    movel([0.126018, -1.331569, -2.603647, -0.777173, 1.570796, 1.696815],accel_mss,speed_ms,0,blend_radius_m)
    movel([0.125748, -1.331456, -2.603719, -0.777214, 1.570796, 1.696544],accel_mss,speed_ms,0,blend_radius_m)
    movel([0.125813, -1.331140, -2.603920, -0.777329, 1.570796, 1.696609],accel_mss,speed_ms,0,blend_radius_m)
    movel([0.126327, -1.330807, -2.604132, -0.777450, 1.570796, 1.697124],accel_mss,speed_ms,0,blend_radius_m)
    movel([0.126943, -1.330606, -2.604260, -0.777523, 1.570796, 1.697739],accel_mss,speed_ms,0,blend_radius_m)
    movel([0.128465, -1.330173, -2.604536, -0.777680, 1.570796, 1.699261],accel_mss,speed_ms,0,blend_radius_m)
    speed_ms = 0.003
    movel([0.128465, -1.333596, -2.606105, -0.772688, 1.570796, 1.699261],accel_mss,speed_ms,0,blend_radius_m)
    speed_ms = 0.007
    movel([0.130070, -1.333157, -2.606385, -0.772846, 1.570796, 1.700866],accel_mss,speed_ms,0,blend_radius_m)
    movel([0.130779, -1.333015, -2.606476, -0.772898, 1.570796, 1.701575],accel_mss,speed_ms,0,blend_radius_m)
    movel([0.131107, -1.333043, -2.606458, -0.772888, 1.570796, 1.701903],accel_mss,speed_ms,0,blend_radius_m)
    movel([0.131205, -1.333224, -2.606343, -0.772822, 1.570796, 1.702001],accel_mss,speed_ms,0,blend_radius_m)
    movel([0.131006, -1.333538, -2.606142, -0.772709, 1.570796, 1.701802],accel_mss,speed_ms,0,blend_radius_m)
    movel([0.130299, -1.333839, -2.605950, -0.772600, 1.570796, 1.701096],accel_mss,speed_ms,0,blend_radius_m)
    movel([0.129539, -1.334076, -2.605798, -0.772515, 1.570796, 1.700335],accel_mss,speed_ms,0,blend_radius_m)
    movel([0.128417, -1.334397, -2.605593, -0.772399, 1.570796, 1.699213],accel_mss,speed_ms,0,blend_radius_m)
    movel([0.127106, -1.334758, -2.605362, -0.772269, 1.570796, 1.697903],accel_mss,speed_ms,0,blend_radius_m)
    movel([0.126423, -1.334924, -2.605256, -0.772210, 1.570796, 1.697219],accel_mss,speed_ms,0,blend_radius_m)
    movel([0.126018, -1.334988, -2.605214, -0.772187, 1.570796, 1.696815],accel_mss,speed_ms,0,blend_radius_m)
    movel([0.125748, -1.334876, -2.605286, -0.772227, 1.570796, 1.696544],accel_mss,speed_ms,0,blend_radius_m)
    movel([0.125813, -1.334561, -2.605488, -0.772340, 1.570796, 1.696609],accel_mss,speed_ms,0,blend_radius_m)
    movel([0.126327, -1.334229, -2.605700, -0.772460, 1.570796, 1.697124],accel_mss,speed_ms,0,blend_radius_m)
    movel([0.126943, -1.334028, -2.605829, -0.772532, 1.570796, 1.697739],accel_mss,speed_ms,0,blend_radius_m)
    movel([0.128465, -1.333596, -2.606105, -0.772688, 1.570796, 1.699261],accel_mss,speed_ms,0,blend_radius_m)
    speed_ms = 0.003
    movel([0.128465, -1.320057, -2.599778, -0.792554, 1.570796, 1.699261],accel_mss,speed_ms,0,blend_radius_m)
    speed_ms = 1.000
    movel([0.128465, -1.294201, -2.586731, -0.831457, 1.570796, 1.699261],accel_mss,speed_ms,0,blend_radius_m)
    movel([0.128376, -1.295380, -2.586019, -0.830991, 1.570796, 1.699172],accel_mss,speed_ms,0,blend_radius_m)
    movel([0.128376, -1.321218, -2.599050, -0.792121, 1.570796, 1.699172],accel_mss,speed_ms,0,blend_radius_m)
    speed_ms = 0.003
    movel([0.128376, -1.331325, -2.603802, -0.777262, 1.570796, 1.699172],accel_mss,speed_ms,0,blend_radius_m)
    speed_ms = 0.007
    movel([0.129253, -1.331084, -2.603956, -0.777349, 1.570796, 1.700049],accel_mss,speed_ms,0,blend_radius_m)
    movel([0.130004, -1.330891, -2.604079, -0.777419, 1.570796, 1.700800],accel_mss,speed_ms,0,blend_radius_m)
    movel([0.130651, -1.330733, -2.604179, -0.777477, 1.570796, 1.701447],accel_mss,speed_ms,0,blend_radius_m)
    movel([0.130767, -1.330971, -2.604028, -0.777390, 1.570796, 1.701564],accel_mss,speed_ms,0,blend_radius_m)
    movel([0.130518, -1.331302, -2.603817, -0.777270, 1.570796, 1.701315],accel_mss,speed_ms,0,blend_radius_m)
    movel([0.129889, -1.331600, -2.603627, -0.777162, 1.570796, 1.700686],accel_mss,speed_ms,0,blend_radius_m)
    movel([0.129257, -1.331804, -2.603497, -0.777088, 1.570796, 1.700053],accel_mss,speed_ms,0,blend_radius_m)
    movel([0.128265, -1.332088, -2.603315, -0.776985, 1.570796, 1.699062],accel_mss,speed_ms,0,blend_radius_m)
    movel([0.127097, -1.332410, -2.603110, -0.776869, 1.570796, 1.697893],accel_mss,speed_ms,0,blend_radius_m)
    movel([0.126547, -1.332536, -2.603030, -0.776824, 1.570796, 1.697343],accel_mss,speed_ms,0,blend_radius_m)
    movel([0.126223, -1.332566, -2.603010, -0.776813, 1.570796, 1.697019],accel_mss,speed_ms,0,blend_radius_m)
    movel([0.126005, -1.332511, -2.603046, -0.776833, 1.570796, 1.696802],accel_mss,speed_ms,0,blend_radius_m)
    movel([0.125850, -1.332354, -2.603146, -0.776889, 1.570796, 1.696647],accel_mss,speed_ms,0,blend_radius_m)
    movel([0.126103, -1.332040, -2.603346, -0.777003, 1.570796, 1.696899],accel_mss,speed_ms,0,blend_radius_m)
    movel([0.126548, -1.331872, -2.603454, -0.777064, 1.570796, 1.697344],accel_mss,speed_ms,0,blend_radius_m)
    movel([0.127233, -1.331654, -2.603593, -0.777143, 1.570796, 1.698030],accel_mss,speed_ms,0,blend_radius_m)
    movel([0.128376, -1.331325, -2.603802, -0.777262, 1.570796, 1.699172],accel_mss,speed_ms,0,blend_radius_m)
    speed_ms = 0.003
    movel([0.128376, -1.334746, -2.605370, -0.772274, 1.570796, 1.699172],accel_mss,speed_ms,0,blend_radius_m)
    speed_ms = 0.007
    movel([0.129253, -1.334505, -2.605524, -0.772360, 1.570796, 1.700049],accel_mss,speed_ms,0,blend_radius_m)
    movel([0.130004, -1.334313, -2.605647, -0.772429, 1.570796, 1.700800],accel_mss,speed_ms,0,blend_radius_m)
    movel([0.130651, -1.334155, -2.605748, -0.772486, 1.570796, 1.701447],accel_mss,speed_ms,0,blend_radius_m)
    movel([0.130767, -1.334392, -2.605596, -0.772401, 1.570796, 1.701564],accel_mss,speed_ms,0,blend_radius_m)
    movel([0.130518, -1.334723, -2.605384, -0.772282, 1.570796, 1.701315],accel_mss,speed_ms,0,blend_radius_m)
    movel([0.129889, -1.335019, -2.605194, -0.772175, 1.570796, 1.700686],accel_mss,speed_ms,0,blend_radius_m)
    movel([0.129257, -1.335223, -2.605064, -0.772102, 1.570796, 1.700053],accel_mss,speed_ms,0,blend_radius_m)
    movel([0.128265, -1.335507, -2.604882, -0.772001, 1.570796, 1.699062],accel_mss,speed_ms,0,blend_radius_m)
    movel([0.127097, -1.335828, -2.604676, -0.771886, 1.570796, 1.697893],accel_mss,speed_ms,0,blend_radius_m)
    movel([0.126547, -1.335953, -2.604595, -0.771841, 1.570796, 1.697343],accel_mss,speed_ms,0,blend_radius_m)
    movel([0.126223, -1.335984, -2.604575, -0.771830, 1.570796, 1.697019],accel_mss,speed_ms,0,blend_radius_m)
    movel([0.126005, -1.335928, -2.604611, -0.771850, 1.570796, 1.696802],accel_mss,speed_ms,0,blend_radius_m)
    movel([0.125850, -1.335772, -2.604711, -0.771906, 1.570796, 1.696647],accel_mss,speed_ms,0,blend_radius_m)
    movel([0.126103, -1.335458, -2.604913, -0.772018, 1.570796, 1.696899],accel_mss,speed_ms,0,blend_radius_m)
    movel([0.126548, -1.335291, -2.605020, -0.772078, 1.570796, 1.697344],accel_mss,speed_ms,0,blend_radius_m)
    movel([0.127233, -1.335073, -2.605160, -0.772156, 1.570796, 1.698030],accel_mss,speed_ms,0,blend_radius_m)
    movel([0.128376, -1.334746, -2.605370, -0.772274, 1.570796, 1.699172],accel_mss,speed_ms,0,blend_radius_m)
    speed_ms = 0.003
    movel([0.128376, -1.321218, -2.599050, -0.792121, 1.570796, 1.699172],accel_mss,speed_ms,0,blend_radius_m)
    speed_ms = 1.000
    movel([0.128376, -1.295380, -2.586019, -0.830991, 1.570796, 1.699172],accel_mss,speed_ms,0,blend_radius_m)
    movel([0.137370, -1.284877, -2.592306, -0.835206, 1.570796, 1.708167],accel_mss,speed_ms,0,blend_radius_m)
    movel([0.137370, -1.310875, -2.605474, -0.796040, 1.570796, 1.708167],accel_mss,speed_ms,0,blend_radius_m)
    speed_ms = 0.003
    movel([0.137370, -1.321053, -2.610278, -0.781058, 1.570796, 1.708167],accel_mss,speed_ms,0,blend_radius_m)
    speed_ms = 0.007
    movel([0.137150, -1.320787, -2.610444, -0.781158, 1.570796, 1.707947],accel_mss,speed_ms,0,blend_radius_m)
    movel([0.137050, -1.320593, -2.610565, -0.781231, 1.570796, 1.707846],accel_mss,speed_ms,0,blend_radius_m)
    movel([0.136937, -1.320377, -2.610700, -0.781312, 1.570796, 1.707734],accel_mss,speed_ms,0,blend_radius_m)
    movel([0.136779, -1.320160, -2.610835, -0.781394, 1.570796, 1.707575],accel_mss,speed_ms,0,blend_radius_m)
    movel([0.136602, -1.319973, -2.610951, -0.781465, 1.570796, 1.707399],accel_mss,speed_ms,0,blend_radius_m)
    movel([0.136439, -1.319851, -2.611027, -0.781511, 1.570796, 1.707236],accel_mss,speed_ms,0,blend_radius_m)
    movel([0.136172, -1.319653, -2.611150, -0.781586, 1.570796, 1.706969],accel_mss,speed_ms,0,blend_radius_m)
    movel([0.136089, -1.319461, -2.611270, -0.781659, 1.570796, 1.706885],accel_mss,speed_ms,0,blend_radius_m)
    movel([0.136418, -1.319173, -2.611448, -0.781767, 1.570796, 1.707214],accel_mss,speed_ms,0,blend_radius_m)
    movel([0.136698, -1.319168, -2.611451, -0.781769, 1.570796, 1.707494],accel_mss,speed_ms,0,blend_radius_m)
    movel([0.136998, -1.319314, -2.611361, -0.781714, 1.570796, 1.707795],accel_mss,speed_ms,0,blend_radius_m)
    movel([0.137280, -1.319584, -2.611193, -0.781612, 1.570796, 1.708076],accel_mss,speed_ms,0,blend_radius_m)
    movel([0.137517, -1.319956, -2.610962, -0.781471, 1.570796, 1.708313],accel_mss,speed_ms,0,blend_radius_m)
    movel([0.137645, -1.320303, -2.610746, -0.781340, 1.570796, 1.708441],accel_mss,speed_ms,0,blend_radius_m)
    movel([0.137672, -1.320655, -2.610527, -0.781207, 1.570796, 1.708469],accel_mss,speed_ms,0,blend_radius_m)
    movel([0.137604, -1.320928, -2.610356, -0.781105, 1.570796, 1.708401],accel_mss,speed_ms,0,blend_radius_m)
    speed_ms = 0.003
    movel([0.137370, -1.324498, -2.611863, -0.776028, 1.570796, 1.708167],accel_mss,speed_ms,0,blend_radius_m)
    speed_ms = 0.007
    movel([0.137150, -1.324233, -2.612030, -0.776127, 1.570796, 1.707947],accel_mss,speed_ms,0,blend_radius_m)
    movel([0.137050, -1.324039, -2.612151, -0.776199, 1.570796, 1.707846],accel_mss,speed_ms,0,blend_radius_m)
    movel([0.136937, -1.323823, -2.612286, -0.776280, 1.570796, 1.707734],accel_mss,speed_ms,0,blend_radius_m)
    movel([0.136779, -1.323607, -2.612421, -0.776361, 1.570796, 1.707575],accel_mss,speed_ms,0,blend_radius_m)
    movel([0.136602, -1.323421, -2.612538, -0.776431, 1.570796, 1.707399],accel_mss,speed_ms,0,blend_radius_m)
    movel([0.136439, -1.323299, -2.612614, -0.776476, 1.570796, 1.707236],accel_mss,speed_ms,0,blend_radius_m)
    movel([0.136172, -1.323102, -2.612737, -0.776550, 1.570796, 1.706969],accel_mss,speed_ms,0,blend_radius_m)
    movel([0.136089, -1.322910, -2.612857, -0.776622, 1.570796, 1.706885],accel_mss,speed_ms,0,blend_radius_m)
    movel([0.136418, -1.322623, -2.613036, -0.776730, 1.570796, 1.707214],accel_mss,speed_ms,0,blend_radius_m)
    movel([0.136698, -1.322618, -2.613039, -0.776732, 1.570796, 1.707494],accel_mss,speed_ms,0,blend_radius_m)
    movel([0.136998, -1.322763, -2.612949, -0.776677, 1.570796, 1.707795],accel_mss,speed_ms,0,blend_radius_m)
    movel([0.137280, -1.323032, -2.612780, -0.776576, 1.570796, 1.708076],accel_mss,speed_ms,0,blend_radius_m)
    movel([0.137517, -1.323403, -2.612549, -0.776437, 1.570796, 1.708313],accel_mss,speed_ms,0,blend_radius_m)
    movel([0.137645, -1.323750, -2.612332, -0.776307, 1.570796, 1.708441],accel_mss,speed_ms,0,blend_radius_m)
    movel([0.137672, -1.324101, -2.612112, -0.776176, 1.570796, 1.708469],accel_mss,speed_ms,0,blend_radius_m)
    movel([0.137604, -1.324374, -2.611941, -0.776074, 1.570796, 1.708401],accel_mss,speed_ms,0,blend_radius_m)
    speed_ms = 0.003
    movel([0.137370, -1.310875, -2.605474, -0.796040, 1.570796, 1.708167],accel_mss,speed_ms,0,blend_radius_m)
    speed_ms = 1.000
    movel([0.137370, -1.284877, -2.592306, -0.835206, 1.570796, 1.708167],accel_mss,speed_ms,0,blend_radius_m)
    movel([0.119252, -1.286116, -2.591572, -0.834701, 1.570796, 1.690048],accel_mss,speed_ms,0,blend_radius_m)
    movel([0.119252, -1.312095, -2.604724, -0.795570, 1.570796, 1.690048],accel_mss,speed_ms,0,blend_radius_m)
    speed_ms = 0.003
    movel([0.119252, -1.322265, -2.609522, -0.780602, 1.570796, 1.690048],accel_mss,speed_ms,0,blend_radius_m)
    speed_ms = 0.007
    movel([0.118849, -1.322907, -2.609120, -0.780362, 1.570796, 1.689646],accel_mss,speed_ms,0,blend_radius_m)
    movel([0.118412, -1.323261, -2.608898, -0.780230, 1.570796, 1.689208],accel_mss,speed_ms,0,blend_radius_m)
    movel([0.117913, -1.323478, -2.608762, -0.780148, 1.570796, 1.688709],accel_mss,speed_ms,0,blend_radius_m)
    movel([0.117430, -1.323523, -2.608734, -0.780132, 1.570796, 1.688226],accel_mss,speed_ms,0,blend_radius_m)
    movel([0.117037, -1.323388, -2.608819, -0.780182, 1.570796, 1.687833],accel_mss,speed_ms,0,blend_radius_m)
    movel([0.116818, -1.323180, -2.608949, -0.780260, 1.570796, 1.687614],accel_mss,speed_ms,0,blend_radius_m)
    movel([0.116741, -1.322943, -2.609098, -0.780349, 1.570796, 1.687538],accel_mss,speed_ms,0,blend_radius_m)
    movel([0.116801, -1.322647, -2.609283, -0.780459, 1.570796, 1.687597],accel_mss,speed_ms,0,blend_radius_m)
    movel([0.117008, -1.322246, -2.609533, -0.780609, 1.570796, 1.687805],accel_mss,speed_ms,0,blend_radius_m)
    movel([0.117254, -1.321909, -2.609744, -0.780736, 1.570796, 1.688050],accel_mss,speed_ms,0,blend_radius_m)
    movel([0.117529, -1.321654, -2.609903, -0.780831, 1.570796, 1.688326],accel_mss,speed_ms,0,blend_radius_m)
    movel([0.117861, -1.321458, -2.610026, -0.780905, 1.570796, 1.688658],accel_mss,speed_ms,0,blend_radius_m)
    movel([0.118286, -1.321301, -2.610124, -0.780964, 1.570796, 1.689083],accel_mss,speed_ms,0,blend_radius_m)
    movel([0.118909, -1.321295, -2.610127, -0.780966, 1.570796, 1.689706],accel_mss,speed_ms,0,blend_radius_m)
    movel([0.119272, -1.321659, -2.609900, -0.780830, 1.570796, 1.690068],accel_mss,speed_ms,0,blend_radius_m)
    movel([0.119252, -1.322265, -2.609522, -0.780602, 1.570796, 1.690048],accel_mss,speed_ms,0,blend_radius_m)
    speed_ms = 0.003
    movel([0.119252, -1.325707, -2.611104, -0.775577, 1.570796, 1.690048],accel_mss,speed_ms,0,blend_radius_m)
    speed_ms = 0.007
    movel([0.118849, -1.326348, -2.610701, -0.775339, 1.570796, 1.689646],accel_mss,speed_ms,0,blend_radius_m)
    movel([0.118412, -1.326701, -2.610479, -0.775209, 1.570796, 1.689208],accel_mss,speed_ms,0,blend_radius_m)
    movel([0.117913, -1.326918, -2.610343, -0.775128, 1.570796, 1.688709],accel_mss,speed_ms,0,blend_radius_m)
    movel([0.117430, -1.326962, -2.610315, -0.775112, 1.570796, 1.688226],accel_mss,speed_ms,0,blend_radius_m)
    movel([0.117037, -1.326828, -2.610399, -0.775162, 1.570796, 1.687833],accel_mss,speed_ms,0,blend_radius_m)
    movel([0.116818, -1.326620, -2.610530, -0.775239, 1.570796, 1.687614],accel_mss,speed_ms,0,blend_radius_m)
    movel([0.116741, -1.326383, -2.610679, -0.775326, 1.570796, 1.687538],accel_mss,speed_ms,0,blend_radius_m)
    movel([0.116801, -1.326089, -2.610865, -0.775436, 1.570796, 1.687597],accel_mss,speed_ms,0,blend_radius_m)
    movel([0.117008, -1.325689, -2.611116, -0.775584, 1.570796, 1.687805],accel_mss,speed_ms,0,blend_radius_m)
    movel([0.117254, -1.325352, -2.611327, -0.775709, 1.570796, 1.688050],accel_mss,speed_ms,0,blend_radius_m)
    movel([0.117529, -1.325098, -2.611487, -0.775804, 1.570796, 1.688326],accel_mss,speed_ms,0,blend_radius_m)
    movel([0.117861, -1.324902, -2.611610, -0.775877, 1.570796, 1.688658],accel_mss,speed_ms,0,blend_radius_m)
    movel([0.118286, -1.324745, -2.611708, -0.775935, 1.570796, 1.689083],accel_mss,speed_ms,0,blend_radius_m)
    movel([0.118909, -1.324740, -2.611712, -0.775937, 1.570796, 1.689706],accel_mss,speed_ms,0,blend_radius_m)
    movel([0.119272, -1.325103, -2.611484, -0.775802, 1.570796, 1.690068],accel_mss,speed_ms,0,blend_radius_m)
    movel([0.119252, -1.325707, -2.611104, -0.775577, 1.570796, 1.690048],accel_mss,speed_ms,0,blend_radius_m)
    speed_ms = 0.003
    movel([0.119252, -1.312095, -2.604724, -0.795570, 1.570796, 1.690048],accel_mss,speed_ms,0,blend_radius_m)
    speed_ms = 1.000
    movel([0.119252, -1.286116, -2.591572, -0.834701, 1.570796, 1.690048],accel_mss,speed_ms,0,blend_radius_m)
    movel([0.117157, -1.287840, -2.590547, -0.834003, 1.570796, 1.687953],accel_mss,speed_ms,0,blend_radius_m)
    movel([0.117157, -1.313793, -2.603676, -0.794920, 1.570796, 1.687953],accel_mss,speed_ms,0,blend_radius_m)
    speed_ms = 0.003
    movel([0.117157, -1.323951, -2.608466, -0.779972, 1.570796, 1.687953],accel_mss,speed_ms,0,blend_radius_m)
    speed_ms = 0.007
    movel([0.116199, -1.324445, -2.608156, -0.779788, 1.570796, 1.686995],accel_mss,speed_ms,0,blend_radius_m)
    movel([0.114974, -1.324825, -2.607917, -0.779647, 1.570796, 1.685771],accel_mss,speed_ms,0,blend_radius_m)
    movel([0.112987, -1.325414, -2.607546, -0.779429, 1.570796, 1.683784],accel_mss,speed_ms,0,blend_radius_m)
    movel([0.109916, -1.326292, -2.606993, -0.779104, 1.570796, 1.680712],accel_mss,speed_ms,0,blend_radius_m)
    movel([0.107439, -1.326950, -2.606578, -0.778861, 1.570796, 1.678235],accel_mss,speed_ms,0,blend_radius_m)
    movel([0.105467, -1.327427, -2.606276, -0.778685, 1.570796, 1.676263],accel_mss,speed_ms,0,blend_radius_m)
    movel([0.105026, -1.327400, -2.606293, -0.778695, 1.570796, 1.675823],accel_mss,speed_ms,0,blend_radius_m)
    movel([0.104891, -1.327141, -2.606457, -0.778791, 1.570796, 1.675687],accel_mss,speed_ms,0,blend_radius_m)
    movel([0.105029, -1.326049, -2.607146, -0.779194, 1.570796, 1.675825],accel_mss,speed_ms,0,blend_radius_m)
    movel([0.105231, -1.324940, -2.607844, -0.779604, 1.570796, 1.676027],accel_mss,speed_ms,0,blend_radius_m)
    movel([0.105466, -1.324531, -2.608101, -0.779756, 1.570796, 1.676262],accel_mss,speed_ms,0,blend_radius_m)
    movel([0.106094, -1.324229, -2.608291, -0.779869, 1.570796, 1.676890],accel_mss,speed_ms,0,blend_radius_m)
    movel([0.106784, -1.324020, -2.608423, -0.779947, 1.570796, 1.677580],accel_mss,speed_ms,0,blend_radius_m)
    movel([0.108077, -1.323673, -2.608640, -0.780076, 1.570796, 1.678873],accel_mss,speed_ms,0,blend_radius_m)
    movel([0.109244, -1.323357, -2.608838, -0.780194, 1.570796, 1.680040],accel_mss,speed_ms,0,blend_radius_m)
    movel([0.110821, -1.322912, -2.609117, -0.780360, 1.570796, 1.681617],accel_mss,speed_ms,0,blend_radius_m)
    movel([0.112506, -1.322432, -2.609417, -0.780540, 1.570796, 1.683302],accel_mss,speed_ms,0,blend_radius_m)
    movel([0.114052, -1.321979, -2.609700, -0.780709, 1.570796, 1.684848],accel_mss,speed_ms,0,blend_radius_m)
    movel([0.115711, -1.321495, -2.610003, -0.780891, 1.570796, 1.686507],accel_mss,speed_ms,0,blend_radius_m)
    movel([0.116781, -1.321202, -2.610185, -0.781001, 1.570796, 1.687578],accel_mss,speed_ms,0,blend_radius_m)
    movel([0.117553, -1.321008, -2.610307, -0.781075, 1.570796, 1.688350],accel_mss,speed_ms,0,blend_radius_m)
    movel([0.117370, -1.321384, -2.610072, -0.780933, 1.570796, 1.688166],accel_mss,speed_ms,0,blend_radius_m)
    movel([0.116917, -1.321847, -2.609783, -0.780759, 1.570796, 1.687714],accel_mss,speed_ms,0,blend_radius_m)
    movel([0.116638, -1.322230, -2.609543, -0.780615, 1.570796, 1.687434],accel_mss,speed_ms,0,blend_radius_m)
    movel([0.116431, -1.322606, -2.609308, -0.780475, 1.570796, 1.687228],accel_mss,speed_ms,0,blend_radius_m)
    movel([0.116340, -1.322909, -2.609119, -0.780361, 1.570796, 1.687136],accel_mss,speed_ms,0,blend_radius_m)
    movel([0.116371, -1.323202, -2.608935, -0.780252, 1.570796, 1.687167],accel_mss,speed_ms,0,blend_radius_m)
    movel([0.116549, -1.323546, -2.608720, -0.780123, 1.570796, 1.687345],accel_mss,speed_ms,0,blend_radius_m)
    movel([0.116786, -1.323831, -2.608541, -0.780017, 1.570796, 1.687582],accel_mss,speed_ms,0,blend_radius_m)
    movel([0.117009, -1.323908, -2.608492, -0.779988, 1.570796, 1.687805],accel_mss,speed_ms,0,blend_radius_m)
    speed_ms = 0.003
    movel([0.117157, -1.327389, -2.610045, -0.774954, 1.570796, 1.687953],accel_mss,speed_ms,0,blend_radius_m)
    speed_ms = 0.007
    movel([0.116199, -1.327882, -2.609735, -0.774772, 1.570796, 1.686995],accel_mss,speed_ms,0,blend_radius_m)
    movel([0.114974, -1.328261, -2.609495, -0.774633, 1.570796, 1.685771],accel_mss,speed_ms,0,blend_radius_m)
    movel([0.112987, -1.328849, -2.609123, -0.774416, 1.570796, 1.683784],accel_mss,speed_ms,0,blend_radius_m)
    movel([0.109916, -1.329725, -2.608569, -0.774095, 1.570796, 1.680712],accel_mss,speed_ms,0,blend_radius_m)
    movel([0.107439, -1.330381, -2.608153, -0.773855, 1.570796, 1.678235],accel_mss,speed_ms,0,blend_radius_m)
    movel([0.105467, -1.330857, -2.607850, -0.773681, 1.570796, 1.676263],accel_mss,speed_ms,0,blend_radius_m)
    movel([0.105026, -1.330830, -2.607868, -0.773691, 1.570796, 1.675823],accel_mss,speed_ms,0,blend_radius_m)
    movel([0.104891, -1.330571, -2.608032, -0.773786, 1.570796, 1.675687],accel_mss,speed_ms,0,blend_radius_m)
    movel([0.105029, -1.329482, -2.608723, -0.774184, 1.570796, 1.675825],accel_mss,speed_ms,0,blend_radius_m)
    movel([0.105231, -1.328376, -2.609422, -0.774590, 1.570796, 1.676027],accel_mss,speed_ms,0,blend_radius_m)
    movel([0.105466, -1.327968, -2.609680, -0.774741, 1.570796, 1.676262],accel_mss,speed_ms,0,blend_radius_m)
    movel([0.106094, -1.327666, -2.609871, -0.774852, 1.570796, 1.676890],accel_mss,speed_ms,0,blend_radius_m)
    movel([0.106784, -1.327458, -2.610002, -0.774929, 1.570796, 1.677580],accel_mss,speed_ms,0,blend_radius_m)
    movel([0.108077, -1.327112, -2.610220, -0.775057, 1.570796, 1.678873],accel_mss,speed_ms,0,blend_radius_m)
    movel([0.109244, -1.326797, -2.610419, -0.775173, 1.570796, 1.680040],accel_mss,speed_ms,0,blend_radius_m)
    movel([0.110821, -1.326353, -2.610698, -0.775338, 1.570796, 1.681617],accel_mss,speed_ms,0,blend_radius_m)
    movel([0.112506, -1.325874, -2.611000, -0.775515, 1.570796, 1.683302],accel_mss,speed_ms,0,blend_radius_m)
    movel([0.114052, -1.325422, -2.611283, -0.775683, 1.570796, 1.684848],accel_mss,speed_ms,0,blend_radius_m)
    movel([0.115711, -1.324939, -2.611587, -0.775863, 1.570796, 1.686507],accel_mss,speed_ms,0,blend_radius_m)
    movel([0.116781, -1.324647, -2.611770, -0.775972, 1.570796, 1.687578],accel_mss,speed_ms,0,blend_radius_m)
    movel([0.117553, -1.324453, -2.611891, -0.776044, 1.570796, 1.688350],accel_mss,speed_ms,0,blend_radius_m)
    movel([0.117370, -1.324829, -2.611656, -0.775904, 1.570796, 1.688166],accel_mss,speed_ms,0,blend_radius_m)
    movel([0.116917, -1.325290, -2.611367, -0.775732, 1.570796, 1.687714],accel_mss,speed_ms,0,blend_radius_m)
    movel([0.116638, -1.325673, -2.611126, -0.775590, 1.570796, 1.687434],accel_mss,speed_ms,0,blend_radius_m)
    movel([0.116431, -1.326048, -2.610891, -0.775451, 1.570796, 1.687228],accel_mss,speed_ms,0,blend_radius_m)
    movel([0.116340, -1.326349, -2.610701, -0.775339, 1.570796, 1.687136],accel_mss,speed_ms,0,blend_radius_m)
    movel([0.116371, -1.326643, -2.610516, -0.775230, 1.570796, 1.687167],accel_mss,speed_ms,0,blend_radius_m)
    movel([0.116549, -1.326985, -2.610300, -0.775104, 1.570796, 1.687345],accel_mss,speed_ms,0,blend_radius_m)
    movel([0.116786, -1.327270, -2.610121, -0.774998, 1.570796, 1.687582],accel_mss,speed_ms,0,blend_radius_m)
    movel([0.117009, -1.327347, -2.610072, -0.774970, 1.570796, 1.687805],accel_mss,speed_ms,0,blend_radius_m)
    speed_ms = 0.003
    movel([0.117157, -1.313793, -2.603676, -0.794920, 1.570796, 1.687953],accel_mss,speed_ms,0,blend_radius_m)
    speed_ms = 1.000
    movel([0.117157, -1.287840, -2.590547, -0.834003, 1.570796, 1.687953],accel_mss,speed_ms,0,blend_radius_m)
    movel([0.107938, -1.297165, -2.584936, -0.830288, 1.570796, 1.678734],accel_mss,speed_ms,0,blend_radius_m)
    movel([0.107938, -1.322976, -2.597944, -0.791469, 1.570796, 1.678734],accel_mss,speed_ms,0,blend_radius_m)
    speed_ms = 0.003
    movel([0.107938, -1.333071, -2.602688, -0.776631, 1.570796, 1.678734],accel_mss,speed_ms,0,blend_radius_m)
    speed_ms = 0.007
    movel([0.107859, -1.333421, -2.602463, -0.776504, 1.570796, 1.678655],accel_mss,speed_ms,0,blend_radius_m)
    movel([0.107233, -1.333668, -2.602305, -0.776416, 1.570796, 1.678029],accel_mss,speed_ms,0,blend_radius_m)
    movel([0.105707, -1.334134, -2.602006, -0.776248, 1.570796, 1.676504],accel_mss,speed_ms,0,blend_radius_m)
    movel([0.104364, -1.334532, -2.601751, -0.776106, 1.570796, 1.675160],accel_mss,speed_ms,0,blend_radius_m)
    movel([0.103784, -1.334679, -2.601657, -0.776053, 1.570796, 1.674580],accel_mss,speed_ms,0,blend_radius_m)
    movel([0.103487, -1.334714, -2.601634, -0.776040, 1.570796, 1.674283],accel_mss,speed_ms,0,blend_radius_m)
    movel([0.103538, -1.334390, -2.601842, -0.776156, 1.570796, 1.674334],accel_mss,speed_ms,0,blend_radius_m)
    movel([0.104072, -1.334096, -2.602031, -0.776262, 1.570796, 1.674868],accel_mss,speed_ms,0,blend_radius_m)
    movel([0.104931, -1.333766, -2.602242, -0.776380, 1.570796, 1.675728],accel_mss,speed_ms,0,blend_radius_m)
    movel([0.106139, -1.333410, -2.602471, -0.776509, 1.570796, 1.676935],accel_mss,speed_ms,0,blend_radius_m)
    movel([0.106867, -1.333221, -2.602591, -0.776576, 1.570796, 1.677664],accel_mss,speed_ms,0,blend_radius_m)
    movel([0.107396, -1.333106, -2.602665, -0.776618, 1.570796, 1.678192],accel_mss,speed_ms,0,blend_radius_m)
    movel([0.107770, -1.333049, -2.602702, -0.776639, 1.570796, 1.678566],accel_mss,speed_ms,0,blend_radius_m)
    speed_ms = 0.003
    movel([0.107938, -1.336487, -2.604252, -0.771650, 1.570796, 1.678734],accel_mss,speed_ms,0,blend_radius_m)
    speed_ms = 0.007
    movel([0.107859, -1.336837, -2.604027, -0.771525, 1.570796, 1.678655],accel_mss,speed_ms,0,blend_radius_m)
    movel([0.107233, -1.337083, -2.603869, -0.771438, 1.570796, 1.678029],accel_mss,speed_ms,0,blend_radius_m)
    movel([0.105707, -1.337548, -2.603569, -0.771272, 1.570796, 1.676504],accel_mss,speed_ms,0,blend_radius_m)
    movel([0.104364, -1.337944, -2.603313, -0.771131, 1.570796, 1.675160],accel_mss,speed_ms,0,blend_radius_m)
    movel([0.103784, -1.338091, -2.603219, -0.771079, 1.570796, 1.674580],accel_mss,speed_ms,0,blend_radius_m)
    movel([0.103487, -1.338126, -2.603196, -0.771067, 1.570796, 1.674283],accel_mss,speed_ms,0,blend_radius_m)
    movel([0.103538, -1.337803, -2.603404, -0.771181, 1.570796, 1.674334],accel_mss,speed_ms,0,blend_radius_m)
    movel([0.104072, -1.337509, -2.603594, -0.771286, 1.570796, 1.674868],accel_mss,speed_ms,0,blend_radius_m)
    movel([0.104931, -1.337181, -2.603806, -0.771403, 1.570796, 1.675728],accel_mss,speed_ms,0,blend_radius_m)
    movel([0.106139, -1.336825, -2.604035, -0.771530, 1.570796, 1.676935],accel_mss,speed_ms,0,blend_radius_m)
    movel([0.106867, -1.336637, -2.604155, -0.771597, 1.570796, 1.677664],accel_mss,speed_ms,0,blend_radius_m)
    movel([0.107396, -1.336522, -2.604229, -0.771637, 1.570796, 1.678192],accel_mss,speed_ms,0,blend_radius_m)
    movel([0.107770, -1.336465, -2.604266, -0.771658, 1.570796, 1.678566],accel_mss,speed_ms,0,blend_radius_m)
    speed_ms = 0.003
    movel([0.107938, -1.322976, -2.597944, -0.791469, 1.570796, 1.678734],accel_mss,speed_ms,0,blend_radius_m)
    speed_ms = 1.000
    movel([0.107938, -1.297165, -2.584936, -0.830288, 1.570796, 1.678734],accel_mss,speed_ms,0,blend_radius_m)
    movel([0.107906, -1.298067, -2.584388, -0.829934, 1.570796, 1.678702],accel_mss,speed_ms,0,blend_radius_m)
    movel([0.107906, -1.323863, -2.597384, -0.791142, 1.570796, 1.678702],accel_mss,speed_ms,0,blend_radius_m)
    speed_ms = 0.003
    movel([0.107906, -1.333952, -2.602123, -0.776314, 1.570796, 1.678702],accel_mss,speed_ms,0,blend_radius_m)
    speed_ms = 0.007
    movel([0.108169, -1.334028, -2.602074, -0.776286, 1.570796, 1.678965],accel_mss,speed_ms,0,blend_radius_m)
    movel([0.108214, -1.334282, -2.601912, -0.776195, 1.570796, 1.679010],accel_mss,speed_ms,0,blend_radius_m)
    movel([0.107800, -1.334603, -2.601706, -0.776080, 1.570796, 1.678597],accel_mss,speed_ms,0,blend_radius_m)
    movel([0.107218, -1.334810, -2.601573, -0.776006, 1.570796, 1.678014],accel_mss,speed_ms,0,blend_radius_m)
    movel([0.105621, -1.335310, -2.601252, -0.775828, 1.570796, 1.676418],accel_mss,speed_ms,0,blend_radius_m)
    movel([0.104231, -1.335734, -2.600979, -0.775676, 1.570796, 1.675027],accel_mss,speed_ms,0,blend_radius_m)
    movel([0.103531, -1.335928, -2.600854, -0.775607, 1.570796, 1.674328],accel_mss,speed_ms,0,blend_radius_m)
    movel([0.103126, -1.336005, -2.600805, -0.775580, 1.570796, 1.673922],accel_mss,speed_ms,0,blend_radius_m)
    movel([0.102888, -1.335886, -2.600881, -0.775622, 1.570796, 1.673684],accel_mss,speed_ms,0,blend_radius_m)
    movel([0.103069, -1.335537, -2.601106, -0.775746, 1.570796, 1.673865],accel_mss,speed_ms,0,blend_radius_m)
    movel([0.103648, -1.335176, -2.601338, -0.775875, 1.570796, 1.674445],accel_mss,speed_ms,0,blend_radius_m)
    movel([0.104251, -1.334968, -2.601471, -0.775950, 1.570796, 1.675047],accel_mss,speed_ms,0,blend_radius_m)
    movel([0.105661, -1.334540, -2.601746, -0.776103, 1.570796, 1.676457],accel_mss,speed_ms,0,blend_radius_m)
    movel([0.107262, -1.334076, -2.602044, -0.776269, 1.570796, 1.678058],accel_mss,speed_ms,0,blend_radius_m)
    movel([0.107906, -1.333952, -2.602123, -0.776314, 1.570796, 1.678702],accel_mss,speed_ms,0,blend_radius_m)
    speed_ms = 0.003
    movel([0.107906, -1.337366, -2.603686, -0.771337, 1.570796, 1.678702],accel_mss,speed_ms,0,blend_radius_m)
    speed_ms = 0.007
    movel([0.108169, -1.337442, -2.603637, -0.771310, 1.570796, 1.678965],accel_mss,speed_ms,0,blend_radius_m)
    movel([0.108214, -1.337695, -2.603474, -0.771220, 1.570796, 1.679010],accel_mss,speed_ms,0,blend_radius_m)
    movel([0.107800, -1.338016, -2.603267, -0.771106, 1.570796, 1.678597],accel_mss,speed_ms,0,blend_radius_m)
    movel([0.107218, -1.338221, -2.603135, -0.771033, 1.570796, 1.678014],accel_mss,speed_ms,0,blend_radius_m)
    movel([0.105621, -1.338720, -2.602813, -0.770856, 1.570796, 1.676418],accel_mss,speed_ms,0,blend_radius_m)
    movel([0.104231, -1.339143, -2.602539, -0.770707, 1.570796, 1.675027],accel_mss,speed_ms,0,blend_radius_m)
    movel([0.103531, -1.339336, -2.602414, -0.770638, 1.570796, 1.674328],accel_mss,speed_ms,0,blend_radius_m)
    movel([0.103126, -1.339413, -2.602364, -0.770611, 1.570796, 1.673922],accel_mss,speed_ms,0,blend_radius_m)
    movel([0.102888, -1.339295, -2.602441, -0.770653, 1.570796, 1.673684],accel_mss,speed_ms,0,blend_radius_m)
    movel([0.103069, -1.338947, -2.602666, -0.770776, 1.570796, 1.673865],accel_mss,speed_ms,0,blend_radius_m)
    movel([0.103648, -1.338586, -2.602899, -0.770904, 1.570796, 1.674445],accel_mss,speed_ms,0,blend_radius_m)
    movel([0.104251, -1.338380, -2.603033, -0.770977, 1.570796, 1.675047],accel_mss,speed_ms,0,blend_radius_m)
    movel([0.105661, -1.337952, -2.603308, -0.771128, 1.570796, 1.676457],accel_mss,speed_ms,0,blend_radius_m)
    movel([0.107262, -1.337490, -2.603607, -0.771293, 1.570796, 1.678058],accel_mss,speed_ms,0,blend_radius_m)
    movel([0.107906, -1.337366, -2.603686, -0.771337, 1.570796, 1.678702],accel_mss,speed_ms,0,blend_radius_m)
    speed_ms = 0.003
    movel([0.107906, -1.323863, -2.597384, -0.791142, 1.570796, 1.678702],accel_mss,speed_ms,0,blend_radius_m)
    speed_ms = 1.000
    movel([0.107906, -1.298067, -2.584388, -0.829934, 1.570796, 1.678702],accel_mss,speed_ms,0,blend_radius_m)
    movel([0.107817, -1.299224, -2.583683, -0.829482, 1.570796, 1.678614],accel_mss,speed_ms,0,blend_radius_m)
    movel([0.107817, -1.325003, -2.596663, -0.790723, 1.570796, 1.678614],accel_mss,speed_ms,0,blend_radius_m)
    speed_ms = 0.003
    movel([0.107817, -1.335084, -2.601397, -0.775908, 1.570796, 1.678614],accel_mss,speed_ms,0,blend_radius_m)
    speed_ms = 0.007
    movel([0.108145, -1.335107, -2.601382, -0.775900, 1.570796, 1.678941],accel_mss,speed_ms,0,blend_radius_m)
    movel([0.108244, -1.335290, -2.601264, -0.775834, 1.570796, 1.679041],accel_mss,speed_ms,0,blend_radius_m)
    movel([0.108029, -1.335613, -2.601057, -0.775719, 1.570796, 1.678825],accel_mss,speed_ms,0,blend_radius_m)
    movel([0.107285, -1.335923, -2.600857, -0.775609, 1.570796, 1.678081],accel_mss,speed_ms,0,blend_radius_m)
    movel([0.106498, -1.336172, -2.600697, -0.775520, 1.570796, 1.677294],accel_mss,speed_ms,0,blend_radius_m)
    movel([0.105363, -1.336503, -2.600484, -0.775402, 1.570796, 1.676160],accel_mss,speed_ms,0,blend_radius_m)
    movel([0.103973, -1.336893, -2.600233, -0.775264, 1.570796, 1.674770],accel_mss,speed_ms,0,blend_radius_m)
    movel([0.103309, -1.337058, -2.600126, -0.775205, 1.570796, 1.674105],accel_mss,speed_ms,0,blend_radius_m)
    movel([0.102936, -1.337114, -2.600090, -0.775185, 1.570796, 1.673733],accel_mss,speed_ms,0,blend_radius_m)
    movel([0.102740, -1.336972, -2.600181, -0.775235, 1.570796, 1.673536],accel_mss,speed_ms,0,blend_radius_m)
    movel([0.102862, -1.336670, -2.600376, -0.775343, 1.570796, 1.673658],accel_mss,speed_ms,0,blend_radius_m)
    movel([0.103469, -1.336343, -2.600587, -0.775459, 1.570796, 1.674266],accel_mss,speed_ms,0,blend_radius_m)
    movel([0.104158, -1.336113, -2.600735, -0.775541, 1.570796, 1.674954],accel_mss,speed_ms,0,blend_radius_m)
    movel([0.105516, -1.335701, -2.601000, -0.775688, 1.570796, 1.676312],accel_mss,speed_ms,0,blend_radius_m)
    movel([0.107118, -1.335235, -2.601300, -0.775854, 1.570796, 1.677914],accel_mss,speed_ms,0,blend_radius_m)
    movel([0.107817, -1.335084, -2.601397, -0.775908, 1.570796, 1.678614],accel_mss,speed_ms,0,blend_radius_m)
    speed_ms = 0.003
    movel([0.107817, -1.338495, -2.602958, -0.770936, 1.570796, 1.678614],accel_mss,speed_ms,0,blend_radius_m)
    speed_ms = 0.007
    movel([0.108145, -1.338518, -2.602943, -0.770928, 1.570796, 1.678941],accel_mss,speed_ms,0,blend_radius_m)
    movel([0.108244, -1.338701, -2.602825, -0.770863, 1.570796, 1.679041],accel_mss,speed_ms,0,blend_radius_m)
    movel([0.108029, -1.339023, -2.602617, -0.770749, 1.570796, 1.678825],accel_mss,speed_ms,0,blend_radius_m)
    movel([0.107285, -1.339332, -2.602417, -0.770640, 1.570796, 1.678081],accel_mss,speed_ms,0,blend_radius_m)
    movel([0.106498, -1.339580, -2.602256, -0.770552, 1.570796, 1.677294],accel_mss,speed_ms,0,blend_radius_m)
    movel([0.105363, -1.339910, -2.602043, -0.770436, 1.570796, 1.676160],accel_mss,speed_ms,0,blend_radius_m)
    movel([0.103973, -1.340299, -2.601791, -0.770299, 1.570796, 1.674770],accel_mss,speed_ms,0,blend_radius_m)
    movel([0.103309, -1.340464, -2.601684, -0.770241, 1.570796, 1.674105],accel_mss,speed_ms,0,blend_radius_m)
    movel([0.102936, -1.340520, -2.601648, -0.770221, 1.570796, 1.673733],accel_mss,speed_ms,0,blend_radius_m)
    movel([0.102740, -1.340379, -2.601739, -0.770271, 1.570796, 1.673536],accel_mss,speed_ms,0,blend_radius_m)
    movel([0.102862, -1.340077, -2.601934, -0.770377, 1.570796, 1.673658],accel_mss,speed_ms,0,blend_radius_m)
    movel([0.103469, -1.339751, -2.602146, -0.770492, 1.570796, 1.674266],accel_mss,speed_ms,0,blend_radius_m)
    movel([0.104158, -1.339521, -2.602295, -0.770573, 1.570796, 1.674954],accel_mss,speed_ms,0,blend_radius_m)
    movel([0.105516, -1.339110, -2.602561, -0.770718, 1.570796, 1.676312],accel_mss,speed_ms,0,blend_radius_m)
    movel([0.107118, -1.338646, -2.602861, -0.770883, 1.570796, 1.677914],accel_mss,speed_ms,0,blend_radius_m)
    movel([0.107817, -1.338495, -2.602958, -0.770936, 1.570796, 1.678614],accel_mss,speed_ms,0,blend_radius_m)
    speed_ms = 0.003
    movel([0.107817, -1.325003, -2.596663, -0.790723, 1.570796, 1.678614],accel_mss,speed_ms,0,blend_radius_m)
    speed_ms = 1.000
    movel([0.107817, -1.299224, -2.583683, -0.829482, 1.570796, 1.678614],accel_mss,speed_ms,0,blend_radius_m)
    movel([0.107647, -1.300433, -2.582945, -0.829012, 1.570796, 1.678443],accel_mss,speed_ms,0,blend_radius_m)
    movel([0.107647, -1.326192, -2.595910, -0.790287, 1.570796, 1.678443],accel_mss,speed_ms,0,blend_radius_m)
    speed_ms = 0.003
    movel([0.107647, -1.336265, -2.600637, -0.775487, 1.570796, 1.678443],accel_mss,speed_ms,0,blend_radius_m)
    speed_ms = 0.007
    movel([0.107997, -1.336268, -2.600635, -0.775486, 1.570796, 1.678793],accel_mss,speed_ms,0,blend_radius_m)
    movel([0.108103, -1.336431, -2.600530, -0.775428, 1.570796, 1.678900],accel_mss,speed_ms,0,blend_radius_m)
    movel([0.107911, -1.336753, -2.600323, -0.775313, 1.570796, 1.678708],accel_mss,speed_ms,0,blend_radius_m)
    movel([0.107201, -1.337066, -2.600121, -0.775202, 1.570796, 1.677997],accel_mss,speed_ms,0,blend_radius_m)
    movel([0.106427, -1.337319, -2.599957, -0.775112, 1.570796, 1.677223],accel_mss,speed_ms,0,blend_radius_m)
    movel([0.105279, -1.337667, -2.599733, -0.774989, 1.570796, 1.676075],accel_mss,speed_ms,0,blend_radius_m)
    movel([0.103926, -1.338063, -2.599477, -0.774849, 1.570796, 1.674722],accel_mss,speed_ms,0,blend_radius_m)
    movel([0.103245, -1.338242, -2.599361, -0.774786, 1.570796, 1.674041],accel_mss,speed_ms,0,blend_radius_m)
    movel([0.102849, -1.338311, -2.599316, -0.774761, 1.570796, 1.673645],accel_mss,speed_ms,0,blend_radius_m)
    movel([0.102612, -1.338193, -2.599393, -0.774803, 1.570796, 1.673408],accel_mss,speed_ms,0,blend_radius_m)
    movel([0.102681, -1.337903, -2.599580, -0.774906, 1.570796, 1.673477],accel_mss,speed_ms,0,blend_radius_m)
    movel([0.103247, -1.337578, -2.599791, -0.775021, 1.570796, 1.674044],accel_mss,speed_ms,0,blend_radius_m)
    movel([0.103920, -1.337343, -2.599942, -0.775104, 1.570796, 1.674716],accel_mss,speed_ms,0,blend_radius_m)
    movel([0.105328, -1.336906, -2.600224, -0.775259, 1.570796, 1.676124],accel_mss,speed_ms,0,blend_radius_m)
    movel([0.106918, -1.336434, -2.600529, -0.775427, 1.570796, 1.677714],accel_mss,speed_ms,0,blend_radius_m)
    movel([0.107647, -1.336265, -2.600637, -0.775487, 1.570796, 1.678443],accel_mss,speed_ms,0,blend_radius_m)
    speed_ms = 0.003
    movel([0.107647, -1.339673, -2.602197, -0.770520, 1.570796, 1.678443],accel_mss,speed_ms,0,blend_radius_m)
    speed_ms = 0.007
    movel([0.107997, -1.339676, -2.602194, -0.770518, 1.570796, 1.678793],accel_mss,speed_ms,0,blend_radius_m)
    movel([0.108103, -1.339838, -2.602089, -0.770461, 1.570796, 1.678900],accel_mss,speed_ms,0,blend_radius_m)
    movel([0.107911, -1.340160, -2.601881, -0.770348, 1.570796, 1.678708],accel_mss,speed_ms,0,blend_radius_m)
    movel([0.107201, -1.340472, -2.601679, -0.770238, 1.570796, 1.677997],accel_mss,speed_ms,0,blend_radius_m)
    movel([0.106427, -1.340725, -2.601515, -0.770149, 1.570796, 1.677223],accel_mss,speed_ms,0,blend_radius_m)
    movel([0.105279, -1.341071, -2.601290, -0.770028, 1.570796, 1.676075],accel_mss,speed_ms,0,blend_radius_m)
    movel([0.103926, -1.341467, -2.601033, -0.769889, 1.570796, 1.674722],accel_mss,speed_ms,0,blend_radius_m)
    movel([0.103245, -1.341645, -2.600917, -0.769827, 1.570796, 1.674041],accel_mss,speed_ms,0,blend_radius_m)
    movel([0.102849, -1.341714, -2.600872, -0.769803, 1.570796, 1.673645],accel_mss,speed_ms,0,blend_radius_m)
    movel([0.102612, -1.341596, -2.600949, -0.769844, 1.570796, 1.673408],accel_mss,speed_ms,0,blend_radius_m)
    movel([0.102681, -1.341307, -2.601137, -0.769945, 1.570796, 1.673477],accel_mss,speed_ms,0,blend_radius_m)
    movel([0.103247, -1.340982, -2.601347, -0.770059, 1.570796, 1.674044],accel_mss,speed_ms,0,blend_radius_m)
    movel([0.103920, -1.340749, -2.601499, -0.770141, 1.570796, 1.674716],accel_mss,speed_ms,0,blend_radius_m)
    movel([0.105328, -1.340312, -2.601782, -0.770294, 1.570796, 1.676124],accel_mss,speed_ms,0,blend_radius_m)
    movel([0.106918, -1.339841, -2.602087, -0.770460, 1.570796, 1.677714],accel_mss,speed_ms,0,blend_radius_m)
    movel([0.107647, -1.339673, -2.602197, -0.770520, 1.570796, 1.678443],accel_mss,speed_ms,0,blend_radius_m)
    speed_ms = 0.003
    movel([0.107647, -1.326192, -2.595910, -0.790287, 1.570796, 1.678443],accel_mss,speed_ms,0,blend_radius_m)
    speed_ms = 1.000
    movel([0.107647, -1.300433, -2.582945, -0.829012, 1.570796, 1.678443],accel_mss,speed_ms,0,blend_radius_m)
    movel([0.107208, -1.301617, -2.582219, -0.828553, 1.570796, 1.678004],accel_mss,speed_ms,0,blend_radius_m)
    movel([0.107208, -1.327358, -2.595169, -0.789862, 1.570796, 1.678004],accel_mss,speed_ms,0,blend_radius_m)
    speed_ms = 0.003
    movel([0.107208, -1.337422, -2.599891, -0.775076, 1.570796, 1.678004],accel_mss,speed_ms,0,blend_radius_m)
    speed_ms = 0.007
    movel([0.107562, -1.337449, -2.599873, -0.775066, 1.570796, 1.678358],accel_mss,speed_ms,0,blend_radius_m)
    movel([0.107604, -1.337704, -2.599709, -0.774976, 1.570796, 1.678401],accel_mss,speed_ms,0,blend_radius_m)
    movel([0.107297, -1.338020, -2.599505, -0.774864, 1.570796, 1.678093],accel_mss,speed_ms,0,blend_radius_m)
    movel([0.106858, -1.338234, -2.599366, -0.774789, 1.570796, 1.677654],accel_mss,speed_ms,0,blend_radius_m)
    movel([0.105706, -1.338626, -2.599113, -0.774650, 1.570796, 1.676502],accel_mss,speed_ms,0,blend_radius_m)
    movel([0.104550, -1.338987, -2.598879, -0.774523, 1.570796, 1.675347],accel_mss,speed_ms,0,blend_radius_m)
    movel([0.103791, -1.339173, -2.598759, -0.774458, 1.570796, 1.674588],accel_mss,speed_ms,0,blend_radius_m)
    movel([0.103264, -1.339241, -2.598714, -0.774434, 1.570796, 1.674060],accel_mss,speed_ms,0,blend_radius_m)
    movel([0.102924, -1.339205, -2.598738, -0.774446, 1.570796, 1.673720],accel_mss,speed_ms,0,blend_radius_m)
    movel([0.102874, -1.338873, -2.598953, -0.774563, 1.570796, 1.673670],accel_mss,speed_ms,0,blend_radius_m)
    movel([0.103227, -1.338630, -2.599110, -0.774649, 1.570796, 1.674023],accel_mss,speed_ms,0,blend_radius_m)
    movel([0.105223, -1.338009, -2.599512, -0.774868, 1.570796, 1.676019],accel_mss,speed_ms,0,blend_radius_m)
    movel([0.107208, -1.337422, -2.599891, -0.775076, 1.570796, 1.678004],accel_mss,speed_ms,0,blend_radius_m)
    speed_ms = 0.003
    movel([0.107208, -1.340828, -2.601448, -0.770113, 1.570796, 1.678004],accel_mss,speed_ms,0,blend_radius_m)
    speed_ms = 0.007
    movel([0.107562, -1.340854, -2.601431, -0.770104, 1.570796, 1.678358],accel_mss,speed_ms,0,blend_radius_m)
    movel([0.107604, -1.341109, -2.601266, -0.770015, 1.570796, 1.678401],accel_mss,speed_ms,0,blend_radius_m)
    movel([0.107297, -1.341424, -2.601061, -0.769904, 1.570796, 1.678093],accel_mss,speed_ms,0,blend_radius_m)
    movel([0.106858, -1.341637, -2.600922, -0.769830, 1.570796, 1.677654],accel_mss,speed_ms,0,blend_radius_m)
    movel([0.105706, -1.342028, -2.600668, -0.769693, 1.570796, 1.676502],accel_mss,speed_ms,0,blend_radius_m)
    movel([0.104550, -1.342388, -2.600434, -0.769567, 1.570796, 1.675347],accel_mss,speed_ms,0,blend_radius_m)
    movel([0.103791, -1.342574, -2.600313, -0.769503, 1.570796, 1.674588],accel_mss,speed_ms,0,blend_radius_m)
    movel([0.103264, -1.342642, -2.600269, -0.769479, 1.570796, 1.674060],accel_mss,speed_ms,0,blend_radius_m)
    movel([0.102924, -1.342605, -2.600292, -0.769491, 1.570796, 1.673720],accel_mss,speed_ms,0,blend_radius_m)
    movel([0.102874, -1.342274, -2.600508, -0.769607, 1.570796, 1.673670],accel_mss,speed_ms,0,blend_radius_m)
    movel([0.103227, -1.342032, -2.600666, -0.769692, 1.570796, 1.674023],accel_mss,speed_ms,0,blend_radius_m)
    movel([0.105223, -1.341412, -2.601068, -0.769908, 1.570796, 1.676019],accel_mss,speed_ms,0,blend_radius_m)
    movel([0.107208, -1.340828, -2.601448, -0.770113, 1.570796, 1.678004],accel_mss,speed_ms,0,blend_radius_m)
    speed_ms = 0.003
    movel([0.107208, -1.327358, -2.595169, -0.789862, 1.570796, 1.678004],accel_mss,speed_ms,0,blend_radius_m)
    speed_ms = 1.000
    movel([0.107208, -1.301617, -2.582219, -0.828553, 1.570796, 1.678004],accel_mss,speed_ms,0,blend_radius_m)
    movel([0.106807, -1.296909, -2.585092, -0.830388, 1.570796, 1.677603],accel_mss,speed_ms,0,blend_radius_m)
    movel([0.106807, -1.322723, -2.598103, -0.791563, 1.570796, 1.677603],accel_mss,speed_ms,0,blend_radius_m)
    speed_ms = 0.003
    movel([0.106807, -1.332820, -2.602848, -0.776721, 1.570796, 1.677603],accel_mss,speed_ms,0,blend_radius_m)
    speed_ms = 0.007
    movel([0.106502, -1.332938, -2.602772, -0.776678, 1.570796, 1.677298],accel_mss,speed_ms,0,blend_radius_m)
    movel([0.105983, -1.333100, -2.602669, -0.776620, 1.570796, 1.676779],accel_mss,speed_ms,0,blend_radius_m)
    movel([0.105487, -1.333239, -2.602580, -0.776570, 1.570796, 1.676283],accel_mss,speed_ms,0,blend_radius_m)
    movel([0.105149, -1.333311, -2.602534, -0.776544, 1.570796, 1.675945],accel_mss,speed_ms,0,blend_radius_m)
    movel([0.104802, -1.333290, -2.602547, -0.776552, 1.570796, 1.675599],accel_mss,speed_ms,0,blend_radius_m)
    movel([0.104798, -1.332989, -2.602740, -0.776660, 1.570796, 1.675594],accel_mss,speed_ms,0,blend_radius_m)
    movel([0.105353, -1.332764, -2.602884, -0.776741, 1.570796, 1.676149],accel_mss,speed_ms,0,blend_radius_m)
    movel([0.106368, -1.332590, -2.602995, -0.776804, 1.570796, 1.677164],accel_mss,speed_ms,0,blend_radius_m)
    movel([0.106788, -1.332536, -2.603029, -0.776823, 1.570796, 1.677584],accel_mss,speed_ms,0,blend_radius_m)
    movel([0.107044, -1.332630, -2.602969, -0.776789, 1.570796, 1.677840],accel_mss,speed_ms,0,blend_radius_m)
    speed_ms = 0.003
    movel([0.106807, -1.336237, -2.604413, -0.771739, 1.570796, 1.677603],accel_mss,speed_ms,0,blend_radius_m)
    speed_ms = 0.007
    movel([0.106502, -1.336354, -2.604337, -0.771697, 1.570796, 1.677298],accel_mss,speed_ms,0,blend_radius_m)
    movel([0.105983, -1.336516, -2.604233, -0.771640, 1.570796, 1.676779],accel_mss,speed_ms,0,blend_radius_m)
    movel([0.105487, -1.336655, -2.604144, -0.771590, 1.570796, 1.676283],accel_mss,speed_ms,0,blend_radius_m)
    movel([0.105149, -1.336727, -2.604098, -0.771565, 1.570796, 1.675945],accel_mss,speed_ms,0,blend_radius_m)
    movel([0.104802, -1.336705, -2.604112, -0.771572, 1.570796, 1.675599],accel_mss,speed_ms,0,blend_radius_m)
    movel([0.104798, -1.336405, -2.604305, -0.771679, 1.570796, 1.675594],accel_mss,speed_ms,0,blend_radius_m)
    movel([0.105353, -1.336181, -2.604449, -0.771759, 1.570796, 1.676149],accel_mss,speed_ms,0,blend_radius_m)
    movel([0.106368, -1.336007, -2.604560, -0.771822, 1.570796, 1.677164],accel_mss,speed_ms,0,blend_radius_m)
    movel([0.106788, -1.335954, -2.604595, -0.771841, 1.570796, 1.677584],accel_mss,speed_ms,0,blend_radius_m)
    movel([0.107044, -1.336047, -2.604534, -0.771807, 1.570796, 1.677840],accel_mss,speed_ms,0,blend_radius_m)
    speed_ms = 0.003
    movel([0.106807, -1.322723, -2.598103, -0.791563, 1.570796, 1.677603],accel_mss,speed_ms,0,blend_radius_m)
    speed_ms = 1.000
    movel([0.106807, -1.296909, -2.585092, -0.830388, 1.570796, 1.677603],accel_mss,speed_ms,0,blend_radius_m)
    movel([0.100351, -1.296361, -2.585424, -0.830604, 1.570796, 1.671147],accel_mss,speed_ms,0,blend_radius_m)
    movel([0.100351, -1.322184, -2.598442, -0.791762, 1.570796, 1.671147],accel_mss,speed_ms,0,blend_radius_m)
    speed_ms = 0.003
    movel([0.100351, -1.332285, -2.603190, -0.776914, 1.570796, 1.671147],accel_mss,speed_ms,0,blend_radius_m)
    speed_ms = 0.007
    movel([0.100080, -1.332260, -2.603206, -0.776923, 1.570796, 1.670877],accel_mss,speed_ms,0,blend_radius_m)
    movel([0.100070, -1.331749, -2.603532, -0.777108, 1.570796, 1.670866],accel_mss,speed_ms,0,blend_radius_m)
    movel([0.099943, -1.331267, -2.603840, -0.777283, 1.570796, 1.670740],accel_mss,speed_ms,0,blend_radius_m)
    movel([0.099742, -1.330807, -2.604133, -0.777450, 1.570796, 1.670539],accel_mss,speed_ms,0,blend_radius_m)
    movel([0.099497, -1.330468, -2.604348, -0.777573, 1.570796, 1.670293],accel_mss,speed_ms,0,blend_radius_m)
    movel([0.099365, -1.330322, -2.604441, -0.777626, 1.570796, 1.670161],accel_mss,speed_ms,0,blend_radius_m)
    movel([0.099182, -1.330081, -2.604594, -0.777714, 1.570796, 1.669978],accel_mss,speed_ms,0,blend_radius_m)
    movel([0.099567, -1.329943, -2.604682, -0.777764, 1.570796, 1.670363],accel_mss,speed_ms,0,blend_radius_m)
    movel([0.100224, -1.329888, -2.604717, -0.777784, 1.570796, 1.671020],accel_mss,speed_ms,0,blend_radius_m)
    movel([0.100489, -1.330079, -2.604595, -0.777714, 1.570796, 1.671285],accel_mss,speed_ms,0,blend_radius_m)
    movel([0.100594, -1.330526, -2.604311, -0.777552, 1.570796, 1.671390],accel_mss,speed_ms,0,blend_radius_m)
    movel([0.100548, -1.331347, -2.603788, -0.777254, 1.570796, 1.671345],accel_mss,speed_ms,0,blend_radius_m)
    movel([0.100488, -1.331853, -2.603466, -0.777070, 1.570796, 1.671284],accel_mss,speed_ms,0,blend_radius_m)
    movel([0.100428, -1.332127, -2.603291, -0.776971, 1.570796, 1.671224],accel_mss,speed_ms,0,blend_radius_m)
    speed_ms = 0.003
    movel([0.100351, -1.335703, -2.604756, -0.771930, 1.570796, 1.671147],accel_mss,speed_ms,0,blend_radius_m)
    speed_ms = 0.007
    movel([0.100080, -1.335678, -2.604772, -0.771939, 1.570796, 1.670877],accel_mss,speed_ms,0,blend_radius_m)
    movel([0.100070, -1.335168, -2.605099, -0.772122, 1.570796, 1.670866],accel_mss,speed_ms,0,blend_radius_m)
    movel([0.099943, -1.334687, -2.605407, -0.772295, 1.570796, 1.670740],accel_mss,speed_ms,0,blend_radius_m)
    movel([0.099742, -1.334228, -2.605701, -0.772460, 1.570796, 1.670539],accel_mss,speed_ms,0,blend_radius_m)
    movel([0.099497, -1.333890, -2.605917, -0.772582, 1.570796, 1.670293],accel_mss,speed_ms,0,blend_radius_m)
    movel([0.099365, -1.333745, -2.606010, -0.772634, 1.570796, 1.670161],accel_mss,speed_ms,0,blend_radius_m)
    movel([0.099182, -1.333504, -2.606164, -0.772721, 1.570796, 1.669978],accel_mss,speed_ms,0,blend_radius_m)
    movel([0.099567, -1.333366, -2.606252, -0.772771, 1.570796, 1.670363],accel_mss,speed_ms,0,blend_radius_m)
    movel([0.100224, -1.333312, -2.606287, -0.772791, 1.570796, 1.671020],accel_mss,speed_ms,0,blend_radius_m)
    movel([0.100489, -1.333503, -2.606165, -0.772722, 1.570796, 1.671285],accel_mss,speed_ms,0,blend_radius_m)
    movel([0.100594, -1.333949, -2.605880, -0.772561, 1.570796, 1.671390],accel_mss,speed_ms,0,blend_radius_m)
    movel([0.100548, -1.334767, -2.605356, -0.772266, 1.570796, 1.671345],accel_mss,speed_ms,0,blend_radius_m)
    movel([0.100488, -1.335272, -2.605032, -0.772085, 1.570796, 1.671284],accel_mss,speed_ms,0,blend_radius_m)
    movel([0.100428, -1.335545, -2.604857, -0.771987, 1.570796, 1.671224],accel_mss,speed_ms,0,blend_radius_m)
    speed_ms = 0.003
    movel([0.100351, -1.322184, -2.598442, -0.791762, 1.570796, 1.671147],accel_mss,speed_ms,0,blend_radius_m)
    speed_ms = 1.000
    movel([0.100351, -1.296361, -2.585424, -0.830604, 1.570796, 1.671147],accel_mss,speed_ms,0,blend_radius_m)
    movel([0.099793, -1.293473, -2.587170, -0.831745, 1.570796, 1.670590],accel_mss,speed_ms,0,blend_radius_m)
    movel([0.099793, -1.319341, -2.600226, -0.792822, 1.570796, 1.670590],accel_mss,speed_ms,0,blend_radius_m)
    speed_ms = 0.003
    movel([0.099793, -1.329461, -2.604988, -0.777940, 1.570796, 1.670590],accel_mss,speed_ms,0,blend_radius_m)
    speed_ms = 0.007
    movel([0.099484, -1.329545, -2.604935, -0.777909, 1.570796, 1.670280],accel_mss,speed_ms,0,blend_radius_m)
    movel([0.099239, -1.329534, -2.604941, -0.777913, 1.570796, 1.670035],accel_mss,speed_ms,0,blend_radius_m)
    movel([0.099173, -1.329280, -2.605103, -0.778006, 1.570796, 1.669969],accel_mss,speed_ms,0,blend_radius_m)
    movel([0.099463, -1.329006, -2.605277, -0.778106, 1.570796, 1.670259],accel_mss,speed_ms,0,blend_radius_m)
    movel([0.099727, -1.328600, -2.605534, -0.778255, 1.570796, 1.670523],accel_mss,speed_ms,0,blend_radius_m)
    movel([0.099806, -1.328310, -2.605718, -0.778361, 1.570796, 1.670603],accel_mss,speed_ms,0,blend_radius_m)
    movel([0.100008, -1.327580, -2.606180, -0.778629, 1.570796, 1.670804],accel_mss,speed_ms,0,blend_radius_m)
    movel([0.100283, -1.326745, -2.606707, -0.778937, 1.570796, 1.671080],accel_mss,speed_ms,0,blend_radius_m)
    movel([0.100572, -1.325975, -2.607193, -0.779221, 1.570796, 1.671369],accel_mss,speed_ms,0,blend_radius_m)
    movel([0.100783, -1.325550, -2.607460, -0.779378, 1.570796, 1.671580],accel_mss,speed_ms,0,blend_radius_m)
    movel([0.101011, -1.325118, -2.607733, -0.779539, 1.570796, 1.671807],accel_mss,speed_ms,0,blend_radius_m)
    movel([0.101399, -1.324234, -2.608288, -0.779867, 1.570796, 1.672195],accel_mss,speed_ms,0,blend_radius_m)
    movel([0.101838, -1.323186, -2.608945, -0.780258, 1.570796, 1.672634],accel_mss,speed_ms,0,blend_radius_m)
    movel([0.102273, -1.322083, -2.609636, -0.780671, 1.570796, 1.673070],accel_mss,speed_ms,0,blend_radius_m)
    movel([0.102450, -1.321652, -2.609904, -0.780832, 1.570796, 1.673246],accel_mss,speed_ms,0,blend_radius_m)
    movel([0.102643, -1.321214, -2.610178, -0.780997, 1.570796, 1.673440],accel_mss,speed_ms,0,blend_radius_m)
    movel([0.102834, -1.320825, -2.610421, -0.781143, 1.570796, 1.673630],accel_mss,speed_ms,0,blend_radius_m)
    movel([0.103093, -1.320382, -2.610696, -0.781310, 1.570796, 1.673889],accel_mss,speed_ms,0,blend_radius_m)
    movel([0.103274, -1.320005, -2.610932, -0.781453, 1.570796, 1.674071],accel_mss,speed_ms,0,blend_radius_m)
    movel([0.103375, -1.319674, -2.611137, -0.781578, 1.570796, 1.674172],accel_mss,speed_ms,0,blend_radius_m)
    movel([0.103705, -1.319383, -2.611318, -0.781688, 1.570796, 1.674501],accel_mss,speed_ms,0,blend_radius_m)
    movel([0.103960, -1.319574, -2.611199, -0.781616, 1.570796, 1.674756],accel_mss,speed_ms,0,blend_radius_m)
    movel([0.103933, -1.319886, -2.611005, -0.781498, 1.570796, 1.674729],accel_mss,speed_ms,0,blend_radius_m)
    movel([0.103783, -1.320327, -2.610731, -0.781331, 1.570796, 1.674579],accel_mss,speed_ms,0,blend_radius_m)
    movel([0.103501, -1.320891, -2.610379, -0.781119, 1.570796, 1.674298],accel_mss,speed_ms,0,blend_radius_m)
    movel([0.103332, -1.321208, -2.610182, -0.780999, 1.570796, 1.674128],accel_mss,speed_ms,0,blend_radius_m)
    movel([0.103182, -1.321516, -2.609990, -0.780883, 1.570796, 1.673978],accel_mss,speed_ms,0,blend_radius_m)
    movel([0.103060, -1.321786, -2.609821, -0.780782, 1.570796, 1.673856],accel_mss,speed_ms,0,blend_radius_m)
    movel([0.102967, -1.322074, -2.609641, -0.780674, 1.570796, 1.673763],accel_mss,speed_ms,0,blend_radius_m)
    movel([0.102824, -1.322435, -2.609416, -0.780539, 1.570796, 1.673620],accel_mss,speed_ms,0,blend_radius_m)
    movel([0.102670, -1.322752, -2.609217, -0.780420, 1.570796, 1.673467],accel_mss,speed_ms,0,blend_radius_m)
    movel([0.102556, -1.323024, -2.609047, -0.780318, 1.570796, 1.673352],accel_mss,speed_ms,0,blend_radius_m)
    movel([0.102484, -1.323290, -2.608880, -0.780219, 1.570796, 1.673280],accel_mss,speed_ms,0,blend_radius_m)
    movel([0.102067, -1.324233, -2.608289, -0.779867, 1.570796, 1.672863],accel_mss,speed_ms,0,blend_radius_m)
    movel([0.101658, -1.325132, -2.607724, -0.779533, 1.570796, 1.672455],accel_mss,speed_ms,0,blend_radius_m)
    movel([0.101394, -1.325660, -2.607392, -0.779338, 1.570796, 1.672190],accel_mss,speed_ms,0,blend_radius_m)
    movel([0.101130, -1.326230, -2.607033, -0.779127, 1.570796, 1.671926],accel_mss,speed_ms,0,blend_radius_m)
    movel([0.100780, -1.327169, -2.606440, -0.778780, 1.570796, 1.671576],accel_mss,speed_ms,0,blend_radius_m)
    movel([0.100468, -1.328096, -2.605853, -0.778440, 1.570796, 1.671264],accel_mss,speed_ms,0,blend_radius_m)
    movel([0.100361, -1.328580, -2.605547, -0.778262, 1.570796, 1.671157],accel_mss,speed_ms,0,blend_radius_m)
    movel([0.100301, -1.328905, -2.605341, -0.778143, 1.570796, 1.671097],accel_mss,speed_ms,0,blend_radius_m)
    movel([0.100218, -1.329160, -2.605179, -0.778050, 1.570796, 1.671014],accel_mss,speed_ms,0,blend_radius_m)
    movel([0.099793, -1.329461, -2.604988, -0.777940, 1.570796, 1.670590],accel_mss,speed_ms,0,blend_radius_m)
    speed_ms = 0.003
    movel([0.099793, -1.332886, -2.606558, -0.772944, 1.570796, 1.670590],accel_mss,speed_ms,0,blend_radius_m)
    speed_ms = 0.007
    movel([0.099484, -1.332970, -2.606505, -0.772914, 1.570796, 1.670280],accel_mss,speed_ms,0,blend_radius_m)
    movel([0.099239, -1.332959, -2.606512, -0.772918, 1.570796, 1.670035],accel_mss,speed_ms,0,blend_radius_m)
    movel([0.099173, -1.332705, -2.606674, -0.773010, 1.570796, 1.669969],accel_mss,speed_ms,0,blend_radius_m)
    movel([0.099463, -1.332432, -2.606848, -0.773109, 1.570796, 1.670259],accel_mss,speed_ms,0,blend_radius_m)
    movel([0.099727, -1.332027, -2.607106, -0.773256, 1.570796, 1.670523],accel_mss,speed_ms,0,blend_radius_m)
    movel([0.099806, -1.331738, -2.607290, -0.773361, 1.570796, 1.670603],accel_mss,speed_ms,0,blend_radius_m)
    movel([0.100008, -1.331009, -2.607754, -0.773626, 1.570796, 1.670804],accel_mss,speed_ms,0,blend_radius_m)
    movel([0.100283, -1.330177, -2.608282, -0.773930, 1.570796, 1.671080],accel_mss,speed_ms,0,blend_radius_m)
    movel([0.100572, -1.329409, -2.608769, -0.774211, 1.570796, 1.671369],accel_mss,speed_ms,0,blend_radius_m)
    movel([0.100783, -1.328985, -2.609038, -0.774367, 1.570796, 1.671580],accel_mss,speed_ms,0,blend_radius_m)
    movel([0.101011, -1.328553, -2.609311, -0.774525, 1.570796, 1.671807],accel_mss,speed_ms,0,blend_radius_m)
    movel([0.101399, -1.327672, -2.609867, -0.774850, 1.570796, 1.672195],accel_mss,speed_ms,0,blend_radius_m)
    movel([0.101838, -1.326626, -2.610526, -0.775236, 1.570796, 1.672634],accel_mss,speed_ms,0,blend_radius_m)
    movel([0.102273, -1.325525, -2.611219, -0.775645, 1.570796, 1.673070],accel_mss,speed_ms,0,blend_radius_m)
    movel([0.102450, -1.325096, -2.611488, -0.775805, 1.570796, 1.673246],accel_mss,speed_ms,0,blend_radius_m)
    movel([0.102643, -1.324659, -2.611762, -0.775967, 1.570796, 1.673440],accel_mss,speed_ms,0,blend_radius_m)
    movel([0.102834, -1.324271, -2.612006, -0.776112, 1.570796, 1.673630],accel_mss,speed_ms,0,blend_radius_m)
    movel([0.103093, -1.323829, -2.612282, -0.776277, 1.570796, 1.673889],accel_mss,speed_ms,0,blend_radius_m)
    movel([0.103274, -1.323452, -2.612518, -0.776419, 1.570796, 1.674071],accel_mss,speed_ms,0,blend_radius_m)
    movel([0.103375, -1.323123, -2.612724, -0.776542, 1.570796, 1.674172],accel_mss,speed_ms,0,blend_radius_m)
    movel([0.103705, -1.322832, -2.612906, -0.776651, 1.570796, 1.674501],accel_mss,speed_ms,0,blend_radius_m)
    movel([0.103960, -1.323023, -2.612787, -0.776580, 1.570796, 1.674756],accel_mss,speed_ms,0,blend_radius_m)
    movel([0.103933, -1.323334, -2.612592, -0.776463, 1.570796, 1.674729],accel_mss,speed_ms,0,blend_radius_m)
    movel([0.103783, -1.323774, -2.612316, -0.776298, 1.570796, 1.674579],accel_mss,speed_ms,0,blend_radius_m)
    movel([0.103501, -1.324337, -2.611965, -0.776088, 1.570796, 1.674298],accel_mss,speed_ms,0,blend_radius_m)
    movel([0.103332, -1.324652, -2.611767, -0.775970, 1.570796, 1.674128],accel_mss,speed_ms,0,blend_radius_m)
    movel([0.103182, -1.324960, -2.611574, -0.775855, 1.570796, 1.673978],accel_mss,speed_ms,0,blend_radius_m)
    movel([0.103060, -1.325229, -2.611405, -0.775755, 1.570796, 1.673856],accel_mss,speed_ms,0,blend_radius_m)
    movel([0.102967, -1.325517, -2.611224, -0.775648, 1.570796, 1.673763],accel_mss,speed_ms,0,blend_radius_m)
    movel([0.102824, -1.325876, -2.610998, -0.775514, 1.570796, 1.673620],accel_mss,speed_ms,0,blend_radius_m)
    movel([0.102670, -1.326194, -2.610799, -0.775397, 1.570796, 1.673467],accel_mss,speed_ms,0,blend_radius_m)
    movel([0.102556, -1.326465, -2.610628, -0.775296, 1.570796, 1.673352],accel_mss,speed_ms,0,blend_radius_m)
    movel([0.102484, -1.326729, -2.610461, -0.775198, 1.570796, 1.673280],accel_mss,speed_ms,0,blend_radius_m)
    movel([0.102067, -1.327671, -2.609868, -0.774850, 1.570796, 1.672863],accel_mss,speed_ms,0,blend_radius_m)
    movel([0.101658, -1.328567, -2.609302, -0.774520, 1.570796, 1.672455],accel_mss,speed_ms,0,blend_radius_m)
    movel([0.101394, -1.329094, -2.608969, -0.774327, 1.570796, 1.672190],accel_mss,speed_ms,0,blend_radius_m)
    movel([0.101130, -1.329662, -2.608609, -0.774118, 1.570796, 1.671926],accel_mss,speed_ms,0,blend_radius_m)
    movel([0.100780, -1.330600, -2.608014, -0.773775, 1.570796, 1.671576],accel_mss,speed_ms,0,blend_radius_m)
    movel([0.100468, -1.331524, -2.607426, -0.773439, 1.570796, 1.671264],accel_mss,speed_ms,0,blend_radius_m)
    movel([0.100361, -1.332007, -2.607119, -0.773263, 1.570796, 1.671157],accel_mss,speed_ms,0,blend_radius_m)
    movel([0.100301, -1.332331, -2.606912, -0.773145, 1.570796, 1.671097],accel_mss,speed_ms,0,blend_radius_m)
    movel([0.100218, -1.332586, -2.606750, -0.773053, 1.570796, 1.671014],accel_mss,speed_ms,0,blend_radius_m)
    movel([0.099793, -1.332886, -2.606558, -0.772944, 1.570796, 1.670590],accel_mss,speed_ms,0,blend_radius_m)
    speed_ms = 0.003
    movel([0.099793, -1.319341, -2.600226, -0.792822, 1.570796, 1.670590],accel_mss,speed_ms,0,blend_radius_m)
    speed_ms = 1.000
    movel([0.099793, -1.293473, -2.587170, -0.831745, 1.570796, 1.670590],accel_mss,speed_ms,0,blend_radius_m)
    movel([0.098466, -1.294527, -2.586534, -0.831328, 1.570796, 1.669263],accel_mss,speed_ms,0,blend_radius_m)
    movel([0.098466, -1.320378, -2.599576, -0.792434, 1.570796, 1.669263],accel_mss,speed_ms,0,blend_radius_m)
    speed_ms = 0.003
    movel([0.098466, -1.330491, -2.604333, -0.777564, 1.570796, 1.669263],accel_mss,speed_ms,0,blend_radius_m)
    speed_ms = 0.007
    movel([0.097937, -1.331191, -2.603888, -0.777310, 1.570796, 1.668733],accel_mss,speed_ms,0,blend_radius_m)
    movel([0.097708, -1.331447, -2.603724, -0.777217, 1.570796, 1.668505],accel_mss,speed_ms,0,blend_radius_m)
    movel([0.097447, -1.331772, -2.603517, -0.777100, 1.570796, 1.668243],accel_mss,speed_ms,0,blend_radius_m)
    movel([0.097197, -1.332112, -2.603300, -0.776977, 1.570796, 1.667993],accel_mss,speed_ms,0,blend_radius_m)
    movel([0.096999, -1.332412, -2.603109, -0.776868, 1.570796, 1.667796],accel_mss,speed_ms,0,blend_radius_m)
    movel([0.096695, -1.332873, -2.602814, -0.776702, 1.570796, 1.667491],accel_mss,speed_ms,0,blend_radius_m)
    movel([0.096384, -1.333007, -2.602728, -0.776654, 1.570796, 1.667180],accel_mss,speed_ms,0,blend_radius_m)
    movel([0.096418, -1.332696, -2.602927, -0.776766, 1.570796, 1.667214],accel_mss,speed_ms,0,blend_radius_m)
    movel([0.096655, -1.332076, -2.603323, -0.776990, 1.570796, 1.667452],accel_mss,speed_ms,0,blend_radius_m)
    movel([0.097107, -1.331352, -2.603785, -0.777252, 1.570796, 1.667903],accel_mss,speed_ms,0,blend_radius_m)
    movel([0.097621, -1.330720, -2.604188, -0.777481, 1.570796, 1.668417],accel_mss,speed_ms,0,blend_radius_m)
    movel([0.098016, -1.330463, -2.604351, -0.777575, 1.570796, 1.668812],accel_mss,speed_ms,0,blend_radius_m)
    movel([0.098367, -1.330396, -2.604394, -0.777599, 1.570796, 1.669163],accel_mss,speed_ms,0,blend_radius_m)
    speed_ms = 0.003
    movel([0.098466, -1.333914, -2.605902, -0.772573, 1.570796, 1.669263],accel_mss,speed_ms,0,blend_radius_m)
    speed_ms = 0.007
    movel([0.097937, -1.334612, -2.605455, -0.772322, 1.570796, 1.668733],accel_mss,speed_ms,0,blend_radius_m)
    movel([0.097708, -1.334867, -2.605291, -0.772230, 1.570796, 1.668505],accel_mss,speed_ms,0,blend_radius_m)
    movel([0.097447, -1.335192, -2.605084, -0.772114, 1.570796, 1.668243],accel_mss,speed_ms,0,blend_radius_m)
    movel([0.097197, -1.335530, -2.604867, -0.771992, 1.570796, 1.667993],accel_mss,speed_ms,0,blend_radius_m)
    movel([0.096999, -1.335830, -2.604674, -0.771885, 1.570796, 1.667796],accel_mss,speed_ms,0,blend_radius_m)
    movel([0.096695, -1.336290, -2.604379, -0.771720, 1.570796, 1.667491],accel_mss,speed_ms,0,blend_radius_m)
    movel([0.096384, -1.336423, -2.604293, -0.771673, 1.570796, 1.667180],accel_mss,speed_ms,0,blend_radius_m)
    movel([0.096418, -1.336113, -2.604492, -0.771784, 1.570796, 1.667214],accel_mss,speed_ms,0,blend_radius_m)
    movel([0.096655, -1.335495, -2.604889, -0.772005, 1.570796, 1.667452],accel_mss,speed_ms,0,blend_radius_m)
    movel([0.097107, -1.334772, -2.605353, -0.772264, 1.570796, 1.667903],accel_mss,speed_ms,0,blend_radius_m)
    movel([0.097621, -1.334141, -2.605756, -0.772491, 1.570796, 1.668417],accel_mss,speed_ms,0,blend_radius_m)
    movel([0.098016, -1.333886, -2.605920, -0.772583, 1.570796, 1.668812],accel_mss,speed_ms,0,blend_radius_m)
    movel([0.098367, -1.333819, -2.605963, -0.772608, 1.570796, 1.669163],accel_mss,speed_ms,0,blend_radius_m)
    speed_ms = 0.003
    movel([0.098466, -1.320378, -2.599576, -0.792434, 1.570796, 1.669263],accel_mss,speed_ms,0,blend_radius_m)
    speed_ms = 1.000
    movel([0.098466, -1.294527, -2.586534, -0.831328, 1.570796, 1.669263],accel_mss,speed_ms,0,blend_radius_m)
    movel([0.086273, -1.300694, -2.582785, -0.828910, 1.570796, 1.657070],accel_mss,speed_ms,0,blend_radius_m)
    movel([0.086273, -1.326449, -2.595747, -0.790193, 1.570796, 1.657070],accel_mss,speed_ms,0,blend_radius_m)
    speed_ms = 0.003
    movel([0.086273, -1.336520, -2.600473, -0.775396, 1.570796, 1.657070],accel_mss,speed_ms,0,blend_radius_m)
    speed_ms = 0.007
    movel([0.086268, -1.336802, -2.600291, -0.775296, 1.570796, 1.657065],accel_mss,speed_ms,0,blend_radius_m)
    movel([0.086058, -1.337141, -2.600072, -0.775175, 1.570796, 1.656855],accel_mss,speed_ms,0,blend_radius_m)
    movel([0.085720, -1.337512, -2.599833, -0.775044, 1.570796, 1.656517],accel_mss,speed_ms,0,blend_radius_m)
    movel([0.085374, -1.337627, -2.599758, -0.775003, 1.570796, 1.656171],accel_mss,speed_ms,0,blend_radius_m)
    movel([0.085224, -1.337395, -2.599909, -0.775086, 1.570796, 1.656020],accel_mss,speed_ms,0,blend_radius_m)
    movel([0.085296, -1.336943, -2.600200, -0.775246, 1.570796, 1.656092],accel_mss,speed_ms,0,blend_radius_m)
    movel([0.085527, -1.336492, -2.600491, -0.775406, 1.570796, 1.656323],accel_mss,speed_ms,0,blend_radius_m)
    movel([0.085833, -1.336264, -2.600638, -0.775487, 1.570796, 1.656630],accel_mss,speed_ms,0,blend_radius_m)
    movel([0.086153, -1.336364, -2.600574, -0.775452, 1.570796, 1.656950],accel_mss,speed_ms,0,blend_radius_m)
    movel([0.086273, -1.336520, -2.600473, -0.775396, 1.570796, 1.657070],accel_mss,speed_ms,0,blend_radius_m)
    speed_ms = 0.003
    movel([0.086273, -1.339927, -2.602032, -0.770430, 1.570796, 1.657070],accel_mss,speed_ms,0,blend_radius_m)
    speed_ms = 0.007
    movel([0.086268, -1.340209, -2.601849, -0.770331, 1.570796, 1.657065],accel_mss,speed_ms,0,blend_radius_m)
    movel([0.086058, -1.340547, -2.601630, -0.770212, 1.570796, 1.656855],accel_mss,speed_ms,0,blend_radius_m)
    movel([0.085720, -1.340917, -2.601390, -0.770082, 1.570796, 1.656517],accel_mss,speed_ms,0,blend_radius_m)
    movel([0.085374, -1.341032, -2.601315, -0.770042, 1.570796, 1.656171],accel_mss,speed_ms,0,blend_radius_m)
    movel([0.085224, -1.340800, -2.601466, -0.770123, 1.570796, 1.656020],accel_mss,speed_ms,0,blend_radius_m)
    movel([0.085296, -1.340349, -2.601758, -0.770282, 1.570796, 1.656092],accel_mss,speed_ms,0,blend_radius_m)
    movel([0.085527, -1.339899, -2.602050, -0.770440, 1.570796, 1.656323],accel_mss,speed_ms,0,blend_radius_m)
    movel([0.085833, -1.339672, -2.602197, -0.770520, 1.570796, 1.656630],accel_mss,speed_ms,0,blend_radius_m)
    movel([0.086153, -1.339772, -2.602133, -0.770485, 1.570796, 1.656950],accel_mss,speed_ms,0,blend_radius_m)
    movel([0.086273, -1.339927, -2.602032, -0.770430, 1.570796, 1.657070],accel_mss,speed_ms,0,blend_radius_m)
    speed_ms = 0.003
    movel([0.086273, -1.326449, -2.595747, -0.790193, 1.570796, 1.657070],accel_mss,speed_ms,0,blend_radius_m)
    speed_ms = 1.000
    movel([0.086273, -1.300694, -2.582785, -0.828910, 1.570796, 1.657070],accel_mss,speed_ms,0,blend_radius_m)
    movel([0.082714, -1.302464, -2.581699, -0.828225, 1.570796, 1.653510],accel_mss,speed_ms,0,blend_radius_m)
    movel([0.082714, -1.328192, -2.594638, -0.789559, 1.570796, 1.653510],accel_mss,speed_ms,0,blend_radius_m)
    speed_ms = 0.003
    movel([0.082714, -1.338250, -2.599356, -0.774783, 1.570796, 1.653510],accel_mss,speed_ms,0,blend_radius_m)
    speed_ms = 0.007
    movel([0.082485, -1.338611, -2.599123, -0.774656, 1.570796, 1.653282],accel_mss,speed_ms,0,blend_radius_m)
    movel([0.082198, -1.338706, -2.599061, -0.774622, 1.570796, 1.652994],accel_mss,speed_ms,0,blend_radius_m)
    movel([0.081704, -1.338685, -2.599075, -0.774630, 1.570796, 1.652501],accel_mss,speed_ms,0,blend_radius_m)
    movel([0.081237, -1.338602, -2.599128, -0.774659, 1.570796, 1.652033],accel_mss,speed_ms,0,blend_radius_m)
    movel([0.081028, -1.338460, -2.599220, -0.774709, 1.570796, 1.651824],accel_mss,speed_ms,0,blend_radius_m)
    movel([0.080976, -1.338247, -2.599358, -0.774784, 1.570796, 1.651773],accel_mss,speed_ms,0,blend_radius_m)
    movel([0.081269, -1.337770, -2.599666, -0.774953, 1.570796, 1.652065],accel_mss,speed_ms,0,blend_radius_m)
    movel([0.081573, -1.337578, -2.599790, -0.775021, 1.570796, 1.652370],accel_mss,speed_ms,0,blend_radius_m)
    movel([0.082083, -1.337514, -2.599831, -0.775043, 1.570796, 1.652880],accel_mss,speed_ms,0,blend_radius_m)
    movel([0.082541, -1.337814, -2.599638, -0.774937, 1.570796, 1.653337],accel_mss,speed_ms,0,blend_radius_m)
    movel([0.082714, -1.338250, -2.599356, -0.774783, 1.570796, 1.653510],accel_mss,speed_ms,0,blend_radius_m)
    speed_ms = 0.003
    movel([0.082714, -1.341653, -2.600912, -0.769824, 1.570796, 1.653510],accel_mss,speed_ms,0,blend_radius_m)
    speed_ms = 0.007
    movel([0.082485, -1.342013, -2.600678, -0.769698, 1.570796, 1.653282],accel_mss,speed_ms,0,blend_radius_m)
    movel([0.082198, -1.342108, -2.600616, -0.769665, 1.570796, 1.652994],accel_mss,speed_ms,0,blend_radius_m)
    movel([0.081704, -1.342087, -2.600630, -0.769672, 1.570796, 1.652501],accel_mss,speed_ms,0,blend_radius_m)
    movel([0.081237, -1.342004, -2.600683, -0.769701, 1.570796, 1.652033],accel_mss,speed_ms,0,blend_radius_m)
    movel([0.081028, -1.341862, -2.600776, -0.769751, 1.570796, 1.651824],accel_mss,speed_ms,0,blend_radius_m)
    movel([0.080976, -1.341651, -2.600913, -0.769825, 1.570796, 1.651773],accel_mss,speed_ms,0,blend_radius_m)
    movel([0.081269, -1.341175, -2.601223, -0.769992, 1.570796, 1.652065],accel_mss,speed_ms,0,blend_radius_m)
    movel([0.081573, -1.340983, -2.601347, -0.770059, 1.570796, 1.652370],accel_mss,speed_ms,0,blend_radius_m)
    movel([0.082083, -1.340919, -2.601389, -0.770081, 1.570796, 1.652880],accel_mss,speed_ms,0,blend_radius_m)
    movel([0.082541, -1.341218, -2.601194, -0.769976, 1.570796, 1.653337],accel_mss,speed_ms,0,blend_radius_m)
    movel([0.082714, -1.341653, -2.600912, -0.769824, 1.570796, 1.653510],accel_mss,speed_ms,0,blend_radius_m)
    speed_ms = 0.003
    movel([0.082714, -1.328192, -2.594638, -0.789559, 1.570796, 1.653510],accel_mss,speed_ms,0,blend_radius_m)
    speed_ms = 1.000
    movel([0.082714, -1.302464, -2.581699, -0.828225, 1.570796, 1.653510],accel_mss,speed_ms,0,blend_radius_m)
    movel([0.083565, -1.303239, -2.581224, -0.827927, 1.570796, 1.654362],accel_mss,speed_ms,0,blend_radius_m)
    movel([0.083565, -1.328954, -2.594152, -0.789283, 1.570796, 1.654362],accel_mss,speed_ms,0,blend_radius_m)
    speed_ms = 0.003
    movel([0.083565, -1.339007, -2.598866, -0.774516, 1.570796, 1.654362],accel_mss,speed_ms,0,blend_radius_m)
    speed_ms = 0.007
    movel([0.083911, -1.338763, -2.599024, -0.774602, 1.570796, 1.654707],accel_mss,speed_ms,0,blend_radius_m)
    movel([0.084285, -1.338774, -2.599017, -0.774598, 1.570796, 1.655081],accel_mss,speed_ms,0,blend_radius_m)
    movel([0.084377, -1.339211, -2.598734, -0.774444, 1.570796, 1.655174],accel_mss,speed_ms,0,blend_radius_m)
    movel([0.084297, -1.339803, -2.598350, -0.774236, 1.570796, 1.655093],accel_mss,speed_ms,0,blend_radius_m)
    movel([0.083981, -1.341688, -2.597124, -0.773577, 1.570796, 1.654778],accel_mss,speed_ms,0,blend_radius_m)
    movel([0.083718, -1.343145, -2.596173, -0.773070, 1.570796, 1.654515],accel_mss,speed_ms,0,blend_radius_m)
    movel([0.083516, -1.343901, -2.595679, -0.772809, 1.570796, 1.654312],accel_mss,speed_ms,0,blend_radius_m)
    movel([0.083313, -1.344244, -2.595455, -0.772690, 1.570796, 1.654109],accel_mss,speed_ms,0,blend_radius_m)
    movel([0.082983, -1.344142, -2.595521, -0.772726, 1.570796, 1.653779],accel_mss,speed_ms,0,blend_radius_m)
    movel([0.083189, -1.341757, -2.597079, -0.773553, 1.570796, 1.653985],accel_mss,speed_ms,0,blend_radius_m)
    movel([0.083413, -1.339401, -2.598611, -0.774377, 1.570796, 1.654209],accel_mss,speed_ms,0,blend_radius_m)
    movel([0.083565, -1.339007, -2.598866, -0.774516, 1.570796, 1.654362],accel_mss,speed_ms,0,blend_radius_m)
    speed_ms = 0.003
    movel([0.083565, -1.342408, -2.600421, -0.769560, 1.570796, 1.654362],accel_mss,speed_ms,0,blend_radius_m)
    speed_ms = 0.007
    movel([0.083911, -1.342165, -2.600579, -0.769645, 1.570796, 1.654707],accel_mss,speed_ms,0,blend_radius_m)
    movel([0.084285, -1.342176, -2.600572, -0.769641, 1.570796, 1.655081],accel_mss,speed_ms,0,blend_radius_m)
    movel([0.084377, -1.342611, -2.600288, -0.769489, 1.570796, 1.655174],accel_mss,speed_ms,0,blend_radius_m)
    movel([0.084297, -1.343203, -2.599903, -0.769283, 1.570796, 1.655093],accel_mss,speed_ms,0,blend_radius_m)
    movel([0.083981, -1.345082, -2.598674, -0.768632, 1.570796, 1.654778],accel_mss,speed_ms,0,blend_radius_m)
    movel([0.083718, -1.346536, -2.597721, -0.768132, 1.570796, 1.654515],accel_mss,speed_ms,0,blend_radius_m)
    movel([0.083516, -1.347290, -2.597226, -0.767874, 1.570796, 1.654312],accel_mss,speed_ms,0,blend_radius_m)
    movel([0.083313, -1.347632, -2.597001, -0.767757, 1.570796, 1.654109],accel_mss,speed_ms,0,blend_radius_m)
    movel([0.082983, -1.347530, -2.597067, -0.767791, 1.570796, 1.653779],accel_mss,speed_ms,0,blend_radius_m)
    movel([0.083189, -1.345152, -2.598629, -0.768608, 1.570796, 1.653985],accel_mss,speed_ms,0,blend_radius_m)
    movel([0.083413, -1.342801, -2.600165, -0.769423, 1.570796, 1.654209],accel_mss,speed_ms,0,blend_radius_m)
    movel([0.083565, -1.342408, -2.600421, -0.769560, 1.570796, 1.654362],accel_mss,speed_ms,0,blend_radius_m)
    speed_ms = 0.003
    movel([0.083565, -1.328954, -2.594152, -0.789283, 1.570796, 1.654362],accel_mss,speed_ms,0,blend_radius_m)
    speed_ms = 1.000
    movel([0.083565, -1.303239, -2.581224, -0.827927, 1.570796, 1.654362],accel_mss,speed_ms,0,blend_radius_m)
    movel([0.083838, -1.302622, -2.581603, -0.828165, 1.570796, 1.654634],accel_mss,speed_ms,0,blend_radius_m)
    movel([0.083838, -1.328347, -2.594539, -0.789503, 1.570796, 1.654634],accel_mss,speed_ms,0,blend_radius_m)
    speed_ms = 0.003
    movel([0.083838, -1.338404, -2.599256, -0.774729, 1.570796, 1.654634],accel_mss,speed_ms,0,blend_radius_m)
    speed_ms = 0.007
    movel([0.083575, -1.338354, -2.599289, -0.774746, 1.570796, 1.654371],accel_mss,speed_ms,0,blend_radius_m)
    movel([0.083364, -1.338238, -2.599364, -0.774787, 1.570796, 1.654160],accel_mss,speed_ms,0,blend_radius_m)
    movel([0.083137, -1.337667, -2.599733, -0.774989, 1.570796, 1.653934],accel_mss,speed_ms,0,blend_radius_m)
    movel([0.082925, -1.337350, -2.599937, -0.775101, 1.570796, 1.653721],accel_mss,speed_ms,0,blend_radius_m)
    movel([0.082638, -1.337145, -2.600070, -0.775174, 1.570796, 1.653434],accel_mss,speed_ms,0,blend_radius_m)
    movel([0.082291, -1.337055, -2.600128, -0.775206, 1.570796, 1.653087],accel_mss,speed_ms,0,blend_radius_m)
    movel([0.081838, -1.337076, -2.600114, -0.775199, 1.570796, 1.652635],accel_mss,speed_ms,0,blend_radius_m)
    movel([0.081455, -1.337176, -2.600050, -0.775163, 1.570796, 1.652252],accel_mss,speed_ms,0,blend_radius_m)
    movel([0.081141, -1.337389, -2.599913, -0.775088, 1.570796, 1.651937],accel_mss,speed_ms,0,blend_radius_m)
    movel([0.080784, -1.337760, -2.599673, -0.774956, 1.570796, 1.651580],accel_mss,speed_ms,0,blend_radius_m)
    movel([0.080489, -1.338156, -2.599417, -0.774816, 1.570796, 1.651285],accel_mss,speed_ms,0,blend_radius_m)
    movel([0.080384, -1.338436, -2.599236, -0.774717, 1.570796, 1.651180],accel_mss,speed_ms,0,blend_radius_m)
    movel([0.080469, -1.338724, -2.599050, -0.774616, 1.570796, 1.651266],accel_mss,speed_ms,0,blend_radius_m)
    movel([0.080802, -1.338966, -2.598892, -0.774530, 1.570796, 1.651598],accel_mss,speed_ms,0,blend_radius_m)
    movel([0.081280, -1.339123, -2.598791, -0.774475, 1.570796, 1.652076],accel_mss,speed_ms,0,blend_radius_m)
    movel([0.081829, -1.339156, -2.598770, -0.774464, 1.570796, 1.652625],accel_mss,speed_ms,0,blend_radius_m)
    movel([0.082528, -1.339181, -2.598753, -0.774455, 1.570796, 1.653324],accel_mss,speed_ms,0,blend_radius_m)
    movel([0.082794, -1.339392, -2.598617, -0.774381, 1.570796, 1.653590],accel_mss,speed_ms,0,blend_radius_m)
    movel([0.082846, -1.339914, -2.598278, -0.774197, 1.570796, 1.653642],accel_mss,speed_ms,0,blend_radius_m)
    movel([0.082677, -1.341845, -2.597022, -0.773522, 1.570796, 1.653473],accel_mss,speed_ms,0,blend_radius_m)
    movel([0.082499, -1.343551, -2.595908, -0.772930, 1.570796, 1.653295],accel_mss,speed_ms,0,blend_radius_m)
    movel([0.082356, -1.344305, -2.595415, -0.772669, 1.570796, 1.653152],accel_mss,speed_ms,0,blend_radius_m)
    movel([0.082163, -1.344704, -2.595153, -0.772532, 1.570796, 1.652960],accel_mss,speed_ms,0,blend_radius_m)
    movel([0.081866, -1.344923, -2.595010, -0.772456, 1.570796, 1.652662],accel_mss,speed_ms,0,blend_radius_m)
    movel([0.081568, -1.344750, -2.595123, -0.772516, 1.570796, 1.652364],accel_mss,speed_ms,0,blend_radius_m)
    movel([0.081509, -1.344436, -2.595329, -0.772624, 1.570796, 1.652305],accel_mss,speed_ms,0,blend_radius_m)
    movel([0.081511, -1.343949, -2.595648, -0.772792, 1.570796, 1.652308],accel_mss,speed_ms,0,blend_radius_m)
    movel([0.081515, -1.343673, -2.595829, -0.772888, 1.570796, 1.652311],accel_mss,speed_ms,0,blend_radius_m)
    movel([0.081498, -1.343418, -2.595995, -0.772976, 1.570796, 1.652294],accel_mss,speed_ms,0,blend_radius_m)
    movel([0.081461, -1.343213, -2.596129, -0.773047, 1.570796, 1.652258],accel_mss,speed_ms,0,blend_radius_m)
    movel([0.081307, -1.343072, -2.596221, -0.773095, 1.570796, 1.652103],accel_mss,speed_ms,0,blend_radius_m)
    movel([0.081039, -1.343053, -2.596234, -0.773102, 1.570796, 1.651836],accel_mss,speed_ms,0,blend_radius_m)
    movel([0.080706, -1.343052, -2.596234, -0.773103, 1.570796, 1.651503],accel_mss,speed_ms,0,blend_radius_m)
    movel([0.080338, -1.343078, -2.596218, -0.773094, 1.570796, 1.651134],accel_mss,speed_ms,0,blend_radius_m)
    movel([0.079939, -1.343105, -2.596200, -0.773084, 1.570796, 1.650735],accel_mss,speed_ms,0,blend_radius_m)
    movel([0.079516, -1.343110, -2.596196, -0.773082, 1.570796, 1.650312],accel_mss,speed_ms,0,blend_radius_m)
    movel([0.079131, -1.343095, -2.596206, -0.773088, 1.570796, 1.649927],accel_mss,speed_ms,0,blend_radius_m)
    movel([0.078857, -1.343061, -2.596229, -0.773099, 1.570796, 1.649653],accel_mss,speed_ms,0,blend_radius_m)
    movel([0.077911, -1.342715, -2.596455, -0.773220, 1.570796, 1.648707],accel_mss,speed_ms,0,blend_radius_m)
    movel([0.077138, -1.342102, -2.596854, -0.773432, 1.570796, 1.647934],accel_mss,speed_ms,0,blend_radius_m)
    movel([0.076602, -1.341277, -2.597392, -0.773720, 1.570796, 1.647398],accel_mss,speed_ms,0,blend_radius_m)
    movel([0.076353, -1.340309, -2.598021, -0.774059, 1.570796, 1.647149],accel_mss,speed_ms,0,blend_radius_m)
    movel([0.076437, -1.339121, -2.598792, -0.774476, 1.570796, 1.647234],accel_mss,speed_ms,0,blend_radius_m)
    movel([0.076894, -1.337754, -2.599676, -0.774958, 1.570796, 1.647690],accel_mss,speed_ms,0,blend_radius_m)
    movel([0.077674, -1.336337, -2.600591, -0.775461, 1.570796, 1.648470],accel_mss,speed_ms,0,blend_radius_m)
    movel([0.078708, -1.335004, -2.601448, -0.775937, 1.570796, 1.649504],accel_mss,speed_ms,0,blend_radius_m)
    movel([0.080811, -1.333153, -2.602635, -0.776601, 1.570796, 1.651607],accel_mss,speed_ms,0,blend_radius_m)
    movel([0.083274, -1.331799, -2.603500, -0.777090, 1.570796, 1.654070],accel_mss,speed_ms,0,blend_radius_m)
    movel([0.085841, -1.331090, -2.603952, -0.777347, 1.570796, 1.656638],accel_mss,speed_ms,0,blend_radius_m)
    movel([0.088231, -1.331107, -2.603941, -0.777341, 1.570796, 1.659028],accel_mss,speed_ms,0,blend_radius_m)
    movel([0.089974, -1.331777, -2.603514, -0.777098, 1.570796, 1.660770],accel_mss,speed_ms,0,blend_radius_m)
    movel([0.091117, -1.333045, -2.602704, -0.776640, 1.570796, 1.661913],accel_mss,speed_ms,0,blend_radius_m)
    movel([0.091521, -1.334728, -2.601626, -0.776036, 1.570796, 1.662317],accel_mss,speed_ms,0,blend_radius_m)
    movel([0.091134, -1.336614, -2.600412, -0.775363, 1.570796, 1.661931],accel_mss,speed_ms,0,blend_radius_m)
    movel([0.090360, -1.338022, -2.599503, -0.774864, 1.570796, 1.661156],accel_mss,speed_ms,0,blend_radius_m)
    movel([0.089237, -1.339332, -2.598656, -0.774402, 1.570796, 1.660033],accel_mss,speed_ms,0,blend_radius_m)
    movel([0.087880, -1.340411, -2.597955, -0.774023, 1.570796, 1.658676],accel_mss,speed_ms,0,blend_radius_m)
    movel([0.086419, -1.341159, -2.597469, -0.773761, 1.570796, 1.657215],accel_mss,speed_ms,0,blend_radius_m)
    movel([0.086085, -1.341294, -2.597381, -0.773714, 1.570796, 1.656881],accel_mss,speed_ms,0,blend_radius_m)
    movel([0.085784, -1.341434, -2.597289, -0.773665, 1.570796, 1.656580],accel_mss,speed_ms,0,blend_radius_m)
    movel([0.085437, -1.341649, -2.597150, -0.773590, 1.570796, 1.656234],accel_mss,speed_ms,0,blend_radius_m)
    movel([0.085272, -1.342062, -2.596880, -0.773446, 1.570796, 1.656068],accel_mss,speed_ms,0,blend_radius_m)
    movel([0.085168, -1.342424, -2.596644, -0.773321, 1.570796, 1.655964],accel_mss,speed_ms,0,blend_radius_m)
    movel([0.085068, -1.342821, -2.596385, -0.773183, 1.570796, 1.655864],accel_mss,speed_ms,0,blend_radius_m)
    movel([0.084872, -1.343546, -2.595911, -0.772931, 1.570796, 1.655669],accel_mss,speed_ms,0,blend_radius_m)
    movel([0.084670, -1.343986, -2.595624, -0.772779, 1.570796, 1.655466],accel_mss,speed_ms,0,blend_radius_m)
    movel([0.084233, -1.344177, -2.595498, -0.772713, 1.570796, 1.655029],accel_mss,speed_ms,0,blend_radius_m)
    movel([0.084159, -1.343630, -2.595857, -0.772903, 1.570796, 1.654955],accel_mss,speed_ms,0,blend_radius_m)
    movel([0.084254, -1.342914, -2.596324, -0.773150, 1.570796, 1.655050],accel_mss,speed_ms,0,blend_radius_m)
    movel([0.084514, -1.341336, -2.597354, -0.773700, 1.570796, 1.655311],accel_mss,speed_ms,0,blend_radius_m)
    movel([0.084702, -1.340274, -2.598044, -0.774071, 1.570796, 1.655498],accel_mss,speed_ms,0,blend_radius_m)
    movel([0.084875, -1.339360, -2.598637, -0.774392, 1.570796, 1.655672],accel_mss,speed_ms,0,blend_radius_m)
    movel([0.085040, -1.338563, -2.599153, -0.774672, 1.570796, 1.655836],accel_mss,speed_ms,0,blend_radius_m)
    movel([0.085311, -1.338276, -2.599339, -0.774774, 1.570796, 1.656107],accel_mss,speed_ms,0,blend_radius_m)
    movel([0.085672, -1.338005, -2.599514, -0.774869, 1.570796, 1.656468],accel_mss,speed_ms,0,blend_radius_m)
    movel([0.086068, -1.337661, -2.599737, -0.774991, 1.570796, 1.656864],accel_mss,speed_ms,0,blend_radius_m)
    movel([0.086444, -1.337219, -2.600022, -0.775148, 1.570796, 1.657240],accel_mss,speed_ms,0,blend_radius_m)
    movel([0.086729, -1.336771, -2.600311, -0.775307, 1.570796, 1.657525],accel_mss,speed_ms,0,blend_radius_m)
    movel([0.086840, -1.336424, -2.600534, -0.775430, 1.570796, 1.657636],accel_mss,speed_ms,0,blend_radius_m)
    movel([0.086756, -1.336163, -2.600703, -0.775523, 1.570796, 1.657553],accel_mss,speed_ms,0,blend_radius_m)
    movel([0.086516, -1.335929, -2.600853, -0.775606, 1.570796, 1.657313],accel_mss,speed_ms,0,blend_radius_m)
    movel([0.085950, -1.335813, -2.600928, -0.775648, 1.570796, 1.656746],accel_mss,speed_ms,0,blend_radius_m)
    movel([0.085372, -1.336061, -2.600768, -0.775559, 1.570796, 1.656169],accel_mss,speed_ms,0,blend_radius_m)
    movel([0.084915, -1.336633, -2.600400, -0.775356, 1.570796, 1.655711],accel_mss,speed_ms,0,blend_radius_m)
    movel([0.084701, -1.337386, -2.599914, -0.775089, 1.570796, 1.655497],accel_mss,speed_ms,0,blend_radius_m)
    movel([0.084629, -1.337702, -2.599710, -0.774977, 1.570796, 1.655425],accel_mss,speed_ms,0,blend_radius_m)
    movel([0.084484, -1.338005, -2.599514, -0.774870, 1.570796, 1.655281],accel_mss,speed_ms,0,blend_radius_m)
    movel([0.084293, -1.338243, -2.599361, -0.774785, 1.570796, 1.655089],accel_mss,speed_ms,0,blend_radius_m)
    movel([0.083838, -1.338404, -2.599256, -0.774729, 1.570796, 1.654634],accel_mss,speed_ms,0,blend_radius_m)
    speed_ms = 0.003
    movel([0.083838, -1.341807, -2.600812, -0.769770, 1.570796, 1.654634],accel_mss,speed_ms,0,blend_radius_m)
    speed_ms = 0.007
    movel([0.083575, -1.341756, -2.600845, -0.769788, 1.570796, 1.654371],accel_mss,speed_ms,0,blend_radius_m)
    movel([0.083364, -1.341641, -2.600920, -0.769828, 1.570796, 1.654160],accel_mss,speed_ms,0,blend_radius_m)
    movel([0.083137, -1.341072, -2.601289, -0.770028, 1.570796, 1.653934],accel_mss,speed_ms,0,blend_radius_m)
    movel([0.082925, -1.340755, -2.601495, -0.770139, 1.570796, 1.653721],accel_mss,speed_ms,0,blend_radius_m)
    movel([0.082638, -1.340551, -2.601627, -0.770210, 1.570796, 1.653434],accel_mss,speed_ms,0,blend_radius_m)
    movel([0.082291, -1.340461, -2.601686, -0.770242, 1.570796, 1.653087],accel_mss,speed_ms,0,blend_radius_m)
    movel([0.081838, -1.340482, -2.601672, -0.770235, 1.570796, 1.652635],accel_mss,speed_ms,0,blend_radius_m)
    movel([0.081455, -1.340581, -2.601608, -0.770200, 1.570796, 1.652252],accel_mss,speed_ms,0,blend_radius_m)
    movel([0.081141, -1.340794, -2.601470, -0.770125, 1.570796, 1.651937],accel_mss,speed_ms,0,blend_radius_m)
    movel([0.080784, -1.341164, -2.601229, -0.769995, 1.570796, 1.651580],accel_mss,speed_ms,0,blend_radius_m)
    movel([0.080489, -1.341559, -2.600973, -0.769857, 1.570796, 1.651285],accel_mss,speed_ms,0,blend_radius_m)
    movel([0.080384, -1.341838, -2.600791, -0.769759, 1.570796, 1.651180],accel_mss,speed_ms,0,blend_radius_m)
    movel([0.080469, -1.342126, -2.600605, -0.769659, 1.570796, 1.651266],accel_mss,speed_ms,0,blend_radius_m)
    movel([0.080802, -1.342368, -2.600447, -0.769574, 1.570796, 1.651598],accel_mss,speed_ms,0,blend_radius_m)
    movel([0.081280, -1.342524, -2.600345, -0.769520, 1.570796, 1.652076],accel_mss,speed_ms,0,blend_radius_m)
    movel([0.081829, -1.342556, -2.600324, -0.769508, 1.570796, 1.652625],accel_mss,speed_ms,0,blend_radius_m)
    movel([0.082528, -1.342582, -2.600308, -0.769500, 1.570796, 1.653324],accel_mss,speed_ms,0,blend_radius_m)
    movel([0.082794, -1.342792, -2.600170, -0.769426, 1.570796, 1.653590],accel_mss,speed_ms,0,blend_radius_m)
    movel([0.082846, -1.343313, -2.599831, -0.769245, 1.570796, 1.653642],accel_mss,speed_ms,0,blend_radius_m)
    movel([0.082677, -1.345239, -2.598572, -0.768578, 1.570796, 1.653473],accel_mss,speed_ms,0,blend_radius_m)
    movel([0.082499, -1.346941, -2.597455, -0.767993, 1.570796, 1.653295],accel_mss,speed_ms,0,blend_radius_m)
    movel([0.082356, -1.347693, -2.596960, -0.767736, 1.570796, 1.653152],accel_mss,speed_ms,0,blend_radius_m)
    movel([0.082163, -1.348091, -2.596698, -0.767600, 1.570796, 1.652960],accel_mss,speed_ms,0,blend_radius_m)
    movel([0.081866, -1.348309, -2.596554, -0.767525, 1.570796, 1.652662],accel_mss,speed_ms,0,blend_radius_m)
    movel([0.081568, -1.348137, -2.596668, -0.767584, 1.570796, 1.652364],accel_mss,speed_ms,0,blend_radius_m)
    movel([0.081509, -1.347824, -2.596874, -0.767691, 1.570796, 1.652305],accel_mss,speed_ms,0,blend_radius_m)
    movel([0.081511, -1.347338, -2.597194, -0.767857, 1.570796, 1.652308],accel_mss,speed_ms,0,blend_radius_m)
    movel([0.081515, -1.347062, -2.597375, -0.767951, 1.570796, 1.652311],accel_mss,speed_ms,0,blend_radius_m)
    movel([0.081498, -1.346808, -2.597542, -0.768038, 1.570796, 1.652294],accel_mss,speed_ms,0,blend_radius_m)
    movel([0.081461, -1.346604, -2.597676, -0.768108, 1.570796, 1.652258],accel_mss,speed_ms,0,blend_radius_m)
    movel([0.081307, -1.346463, -2.597769, -0.768157, 1.570796, 1.652103],accel_mss,speed_ms,0,blend_radius_m)
    movel([0.081039, -1.346444, -2.597782, -0.768163, 1.570796, 1.651836],accel_mss,speed_ms,0,blend_radius_m)
    movel([0.080706, -1.346443, -2.597782, -0.768164, 1.570796, 1.651503],accel_mss,speed_ms,0,blend_radius_m)
    movel([0.080338, -1.346469, -2.597765, -0.768155, 1.570796, 1.651134],accel_mss,speed_ms,0,blend_radius_m)
    movel([0.079939, -1.346496, -2.597748, -0.768146, 1.570796, 1.650735],accel_mss,speed_ms,0,blend_radius_m)
    movel([0.079516, -1.346501, -2.597744, -0.768144, 1.570796, 1.650312],accel_mss,speed_ms,0,blend_radius_m)
    movel([0.079131, -1.346486, -2.597754, -0.768149, 1.570796, 1.649927],accel_mss,speed_ms,0,blend_radius_m)
    movel([0.078857, -1.346452, -2.597776, -0.768161, 1.570796, 1.649653],accel_mss,speed_ms,0,blend_radius_m)
    movel([0.077911, -1.346107, -2.598003, -0.768279, 1.570796, 1.648707],accel_mss,speed_ms,0,blend_radius_m)
    movel([0.077138, -1.345496, -2.598404, -0.768490, 1.570796, 1.647934],accel_mss,speed_ms,0,blend_radius_m)
    movel([0.076602, -1.344673, -2.598942, -0.768774, 1.570796, 1.647398],accel_mss,speed_ms,0,blend_radius_m)
    movel([0.076353, -1.343707, -2.599574, -0.769108, 1.570796, 1.647149],accel_mss,speed_ms,0,blend_radius_m)
    movel([0.076437, -1.342522, -2.600346, -0.769520, 1.570796, 1.647234],accel_mss,speed_ms,0,blend_radius_m)
    movel([0.076894, -1.341159, -2.601233, -0.769997, 1.570796, 1.647690],accel_mss,speed_ms,0,blend_radius_m)
    movel([0.077674, -1.339745, -2.602150, -0.770494, 1.570796, 1.648470],accel_mss,speed_ms,0,blend_radius_m)
    movel([0.078708, -1.338415, -2.603009, -0.770964, 1.570796, 1.649504],accel_mss,speed_ms,0,blend_radius_m)
    movel([0.080811, -1.336569, -2.604199, -0.771621, 1.570796, 1.651607],accel_mss,speed_ms,0,blend_radius_m)
    movel([0.083274, -1.335218, -2.605067, -0.772104, 1.570796, 1.654070],accel_mss,speed_ms,0,blend_radius_m)
    movel([0.085841, -1.334511, -2.605520, -0.772358, 1.570796, 1.656638],accel_mss,speed_ms,0,blend_radius_m)
    movel([0.088231, -1.334527, -2.605509, -0.772352, 1.570796, 1.659028],accel_mss,speed_ms,0,blend_radius_m)
    movel([0.089974, -1.335197, -2.605081, -0.772112, 1.570796, 1.660770],accel_mss,speed_ms,0,blend_radius_m)
    movel([0.091117, -1.336461, -2.604269, -0.771659, 1.570796, 1.661913],accel_mss,speed_ms,0,blend_radius_m)
    movel([0.091521, -1.338140, -2.603187, -0.771062, 1.570796, 1.662317],accel_mss,speed_ms,0,blend_radius_m)
    movel([0.091134, -1.340021, -2.601971, -0.770397, 1.570796, 1.661931],accel_mss,speed_ms,0,blend_radius_m)
    movel([0.090360, -1.341426, -2.601060, -0.769904, 1.570796, 1.661156],accel_mss,speed_ms,0,blend_radius_m)
    movel([0.089237, -1.342732, -2.600210, -0.769447, 1.570796, 1.660033],accel_mss,speed_ms,0,blend_radius_m)
    movel([0.087880, -1.343808, -2.599508, -0.769073, 1.570796, 1.658676],accel_mss,speed_ms,0,blend_radius_m)
    movel([0.086419, -1.344555, -2.599020, -0.768814, 1.570796, 1.657215],accel_mss,speed_ms,0,blend_radius_m)
    movel([0.086085, -1.344690, -2.598932, -0.768768, 1.570796, 1.656881],accel_mss,speed_ms,0,blend_radius_m)
    movel([0.085784, -1.344830, -2.598840, -0.768719, 1.570796, 1.656580],accel_mss,speed_ms,0,blend_radius_m)
    movel([0.085437, -1.345043, -2.598700, -0.768646, 1.570796, 1.656234],accel_mss,speed_ms,0,blend_radius_m)
    movel([0.085272, -1.345456, -2.598430, -0.768503, 1.570796, 1.656068],accel_mss,speed_ms,0,blend_radius_m)
    movel([0.085168, -1.345817, -2.598193, -0.768379, 1.570796, 1.655964],accel_mss,speed_ms,0,blend_radius_m)
    movel([0.085068, -1.346213, -2.597933, -0.768243, 1.570796, 1.655864],accel_mss,speed_ms,0,blend_radius_m)
    movel([0.084872, -1.346936, -2.597458, -0.767995, 1.570796, 1.655669],accel_mss,speed_ms,0,blend_radius_m)
    movel([0.084670, -1.347375, -2.597170, -0.767844, 1.570796, 1.655466],accel_mss,speed_ms,0,blend_radius_m)
    movel([0.084233, -1.347565, -2.597044, -0.767779, 1.570796, 1.655029],accel_mss,speed_ms,0,blend_radius_m)
    movel([0.084159, -1.347019, -2.597404, -0.767966, 1.570796, 1.654955],accel_mss,speed_ms,0,blend_radius_m)
    movel([0.084254, -1.346306, -2.597872, -0.768211, 1.570796, 1.655050],accel_mss,speed_ms,0,blend_radius_m)
    movel([0.084514, -1.344731, -2.598904, -0.768754, 1.570796, 1.655311],accel_mss,speed_ms,0,blend_radius_m)
    movel([0.084702, -1.343673, -2.599596, -0.769120, 1.570796, 1.655498],accel_mss,speed_ms,0,blend_radius_m)
    movel([0.084875, -1.342761, -2.600191, -0.769437, 1.570796, 1.655672],accel_mss,speed_ms,0,blend_radius_m)
    movel([0.085040, -1.341966, -2.600709, -0.769715, 1.570796, 1.655836],accel_mss,speed_ms,0,blend_radius_m)
    movel([0.085311, -1.341679, -2.600895, -0.769815, 1.570796, 1.656107],accel_mss,speed_ms,0,blend_radius_m)
    movel([0.085672, -1.341409, -2.601070, -0.769909, 1.570796, 1.656468],accel_mss,speed_ms,0,blend_radius_m)
    movel([0.086068, -1.341066, -2.601294, -0.770030, 1.570796, 1.656864],accel_mss,speed_ms,0,blend_radius_m)
    movel([0.086444, -1.340624, -2.601580, -0.770185, 1.570796, 1.657240],accel_mss,speed_ms,0,blend_radius_m)
    movel([0.086729, -1.340178, -2.601869, -0.770342, 1.570796, 1.657525],accel_mss,speed_ms,0,blend_radius_m)
    movel([0.086840, -1.339832, -2.602093, -0.770464, 1.570796, 1.657636],accel_mss,speed_ms,0,blend_radius_m)
    movel([0.086756, -1.339572, -2.602262, -0.770555, 1.570796, 1.657553],accel_mss,speed_ms,0,blend_radius_m)
    movel([0.086516, -1.339338, -2.602413, -0.770638, 1.570796, 1.657313],accel_mss,speed_ms,0,blend_radius_m)
    movel([0.085950, -1.339222, -2.602488, -0.770679, 1.570796, 1.656746],accel_mss,speed_ms,0,blend_radius_m)
    movel([0.085372, -1.339470, -2.602328, -0.770591, 1.570796, 1.656169],accel_mss,speed_ms,0,blend_radius_m)
    movel([0.084915, -1.340040, -2.601959, -0.770390, 1.570796, 1.655711],accel_mss,speed_ms,0,blend_radius_m)
    movel([0.084701, -1.340791, -2.601472, -0.770126, 1.570796, 1.655497],accel_mss,speed_ms,0,blend_radius_m)
    movel([0.084629, -1.341106, -2.601267, -0.770016, 1.570796, 1.655425],accel_mss,speed_ms,0,blend_radius_m)
    movel([0.084484, -1.341409, -2.601071, -0.769910, 1.570796, 1.655281],accel_mss,speed_ms,0,blend_radius_m)
    movel([0.084293, -1.341646, -2.600916, -0.769826, 1.570796, 1.655089],accel_mss,speed_ms,0,blend_radius_m)
    movel([0.083838, -1.341807, -2.600812, -0.769770, 1.570796, 1.654634],accel_mss,speed_ms,0,blend_radius_m)
    speed_ms = 0.003
    movel([0.083838, -1.328347, -2.594539, -0.789503, 1.570796, 1.654634],accel_mss,speed_ms,0,blend_radius_m)
    speed_ms = 1.000
    movel([0.083838, -1.302622, -2.581603, -0.828165, 1.570796, 1.654634],accel_mss,speed_ms,0,blend_radius_m)
    movel([0.083131, -1.309400, -2.577409, -0.825580, 1.570796, 1.653928],accel_mss,speed_ms,0,blend_radius_m)
    movel([0.083131, -1.335017, -2.590258, -0.787114, 1.570796, 1.653928],accel_mss,speed_ms,0,blend_radius_m)
    speed_ms = 0.003
    movel([0.083131, -1.345027, -2.594942, -0.772421, 1.570796, 1.653928],accel_mss,speed_ms,0,blend_radius_m)
    speed_ms = 0.007
    movel([0.084912, -1.344646, -2.595191, -0.772552, 1.570796, 1.655708],accel_mss,speed_ms,0,blend_radius_m)
    movel([0.085226, -1.344667, -2.595177, -0.772544, 1.570796, 1.656023],accel_mss,speed_ms,0,blend_radius_m)
    movel([0.085321, -1.344944, -2.594996, -0.772449, 1.570796, 1.656117],accel_mss,speed_ms,0,blend_radius_m)
    movel([0.085214, -1.345307, -2.594758, -0.772325, 1.570796, 1.656010],accel_mss,speed_ms,0,blend_radius_m)
    movel([0.085158, -1.345566, -2.594588, -0.772236, 1.570796, 1.655955],accel_mss,speed_ms,0,blend_radius_m)
    movel([0.085106, -1.345844, -2.594405, -0.772140, 1.570796, 1.655902],accel_mss,speed_ms,0,blend_radius_m)
    movel([0.085067, -1.346106, -2.594233, -0.772050, 1.570796, 1.655864],accel_mss,speed_ms,0,blend_radius_m)
    movel([0.085015, -1.346429, -2.594020, -0.771940, 1.570796, 1.655812],accel_mss,speed_ms,0,blend_radius_m)
    movel([0.084839, -1.346835, -2.593753, -0.771801, 1.570796, 1.655635],accel_mss,speed_ms,0,blend_radius_m)
    movel([0.084290, -1.347303, -2.593444, -0.771641, 1.570796, 1.655087],accel_mss,speed_ms,0,blend_radius_m)
    movel([0.083746, -1.347575, -2.593265, -0.771549, 1.570796, 1.654542],accel_mss,speed_ms,0,blend_radius_m)
    movel([0.083025, -1.347847, -2.593086, -0.771456, 1.570796, 1.653821],accel_mss,speed_ms,0,blend_radius_m)
    movel([0.082091, -1.348128, -2.592900, -0.771361, 1.570796, 1.652888],accel_mss,speed_ms,0,blend_radius_m)
    movel([0.081241, -1.348334, -2.592764, -0.771291, 1.570796, 1.652037],accel_mss,speed_ms,0,blend_radius_m)
    movel([0.080813, -1.348339, -2.592761, -0.771289, 1.570796, 1.651610],accel_mss,speed_ms,0,blend_radius_m)
    movel([0.080675, -1.348167, -2.592874, -0.771347, 1.570796, 1.651471],accel_mss,speed_ms,0,blend_radius_m)
    movel([0.080768, -1.347825, -2.593100, -0.771464, 1.570796, 1.651564],accel_mss,speed_ms,0,blend_radius_m)
    movel([0.080890, -1.347520, -2.593302, -0.771568, 1.570796, 1.651686],accel_mss,speed_ms,0,blend_radius_m)
    movel([0.080645, -1.347327, -2.593429, -0.771633, 1.570796, 1.651441],accel_mss,speed_ms,0,blend_radius_m)
    movel([0.080619, -1.347111, -2.593571, -0.771707, 1.570796, 1.651416],accel_mss,speed_ms,0,blend_radius_m)
    movel([0.080919, -1.346779, -2.593790, -0.771820, 1.570796, 1.651715],accel_mss,speed_ms,0,blend_radius_m)
    movel([0.080769, -1.346426, -2.594022, -0.771941, 1.570796, 1.651566],accel_mss,speed_ms,0,blend_radius_m)
    movel([0.080640, -1.346238, -2.594146, -0.772005, 1.570796, 1.651436],accel_mss,speed_ms,0,blend_radius_m)
    movel([0.080628, -1.346014, -2.594293, -0.772082, 1.570796, 1.651424],accel_mss,speed_ms,0,blend_radius_m)
    movel([0.080942, -1.345606, -2.594561, -0.772222, 1.570796, 1.651739],accel_mss,speed_ms,0,blend_radius_m)
    movel([0.081368, -1.345424, -2.594681, -0.772284, 1.570796, 1.652164],accel_mss,speed_ms,0,blend_radius_m)
    movel([0.083131, -1.345027, -2.594942, -0.772421, 1.570796, 1.653928],accel_mss,speed_ms,0,blend_radius_m)
    speed_ms = 0.003
    movel([0.083131, -1.348413, -2.596486, -0.767490, 1.570796, 1.653928],accel_mss,speed_ms,0,blend_radius_m)
    speed_ms = 0.007
    movel([0.084912, -1.348033, -2.596736, -0.767620, 1.570796, 1.655708],accel_mss,speed_ms,0,blend_radius_m)
    movel([0.085226, -1.348054, -2.596722, -0.767612, 1.570796, 1.656023],accel_mss,speed_ms,0,blend_radius_m)
    movel([0.085321, -1.348330, -2.596541, -0.767518, 1.570796, 1.656117],accel_mss,speed_ms,0,blend_radius_m)
    movel([0.085214, -1.348692, -2.596302, -0.767395, 1.570796, 1.656010],accel_mss,speed_ms,0,blend_radius_m)
    movel([0.085158, -1.348950, -2.596131, -0.767307, 1.570796, 1.655955],accel_mss,speed_ms,0,blend_radius_m)
    movel([0.085106, -1.349228, -2.595948, -0.767213, 1.570796, 1.655902],accel_mss,speed_ms,0,blend_radius_m)
    movel([0.085067, -1.349489, -2.595775, -0.767124, 1.570796, 1.655864],accel_mss,speed_ms,0,blend_radius_m)
    movel([0.085015, -1.349812, -2.595562, -0.767015, 1.570796, 1.655812],accel_mss,speed_ms,0,blend_radius_m)
    movel([0.084839, -1.350216, -2.595294, -0.766878, 1.570796, 1.655635],accel_mss,speed_ms,0,blend_radius_m)
    movel([0.084290, -1.350683, -2.594985, -0.766720, 1.570796, 1.655087],accel_mss,speed_ms,0,blend_radius_m)
    movel([0.083746, -1.350954, -2.594806, -0.766629, 1.570796, 1.654542],accel_mss,speed_ms,0,blend_radius_m)
    movel([0.083025, -1.351226, -2.594626, -0.766538, 1.570796, 1.653821],accel_mss,speed_ms,0,blend_radius_m)
    movel([0.082091, -1.351507, -2.594439, -0.766443, 1.570796, 1.652888],accel_mss,speed_ms,0,blend_radius_m)
    movel([0.081241, -1.351712, -2.594303, -0.766374, 1.570796, 1.652037],accel_mss,speed_ms,0,blend_radius_m)
